NETWORK
TITLE = Set recipe parameters if starting UO_MX_CIP running SUBSTATE
//------------------------------------------------------------------------//
// Set recipe parameters:                                                 //
//------------------------------------------------------------------------//
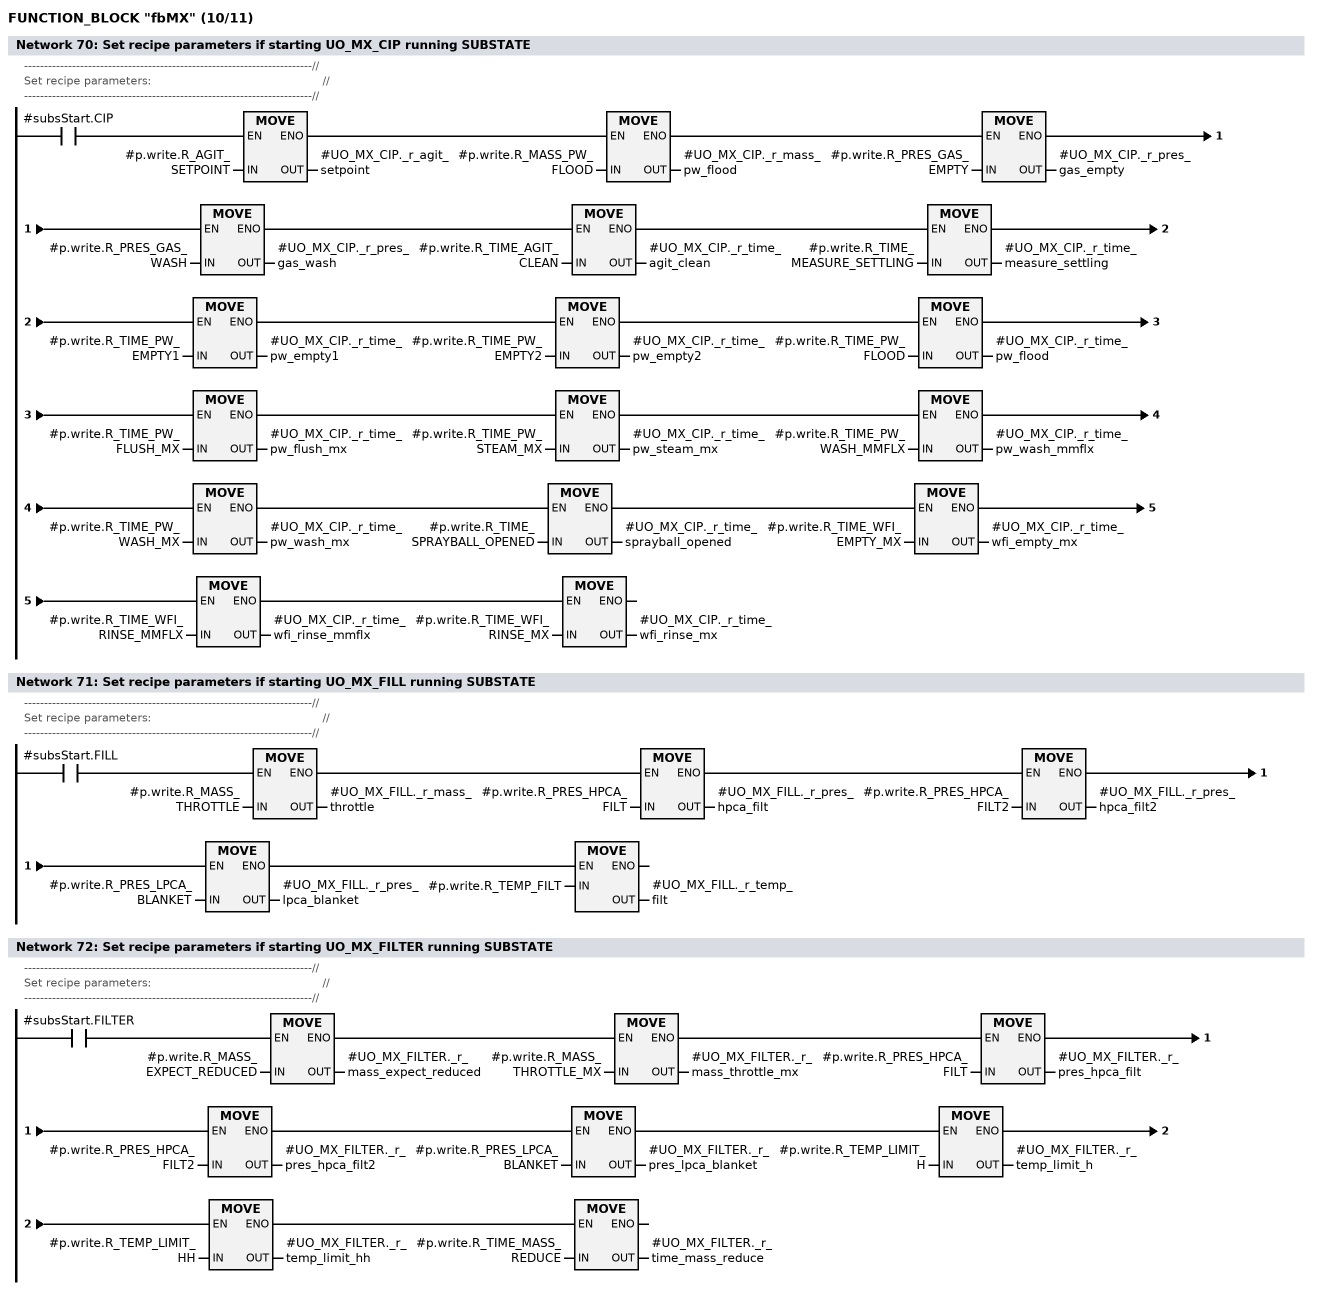
      A #subsStart.CIP;
      JCN _noStaticParms_CIP;
      L #p.write.R_AGIT_SETPOINT;
      T #UO_MX_CIP._r_agit_setpoint;
      L #p.write.R_MASS_PW_FLOOD;
      T #UO_MX_CIP._r_mass_pw_flood;
      L #p.write.R_PRES_GAS_EMPTY;
      T #UO_MX_CIP._r_pres_gas_empty;
      L #p.write.R_PRES_GAS_WASH;
      T #UO_MX_CIP._r_pres_gas_wash;
      L #p.write.R_TIME_AGIT_CLEAN;
      T #UO_MX_CIP._r_time_agit_clean;
      L #p.write.R_TIME_MEASURE_SETTLING;
      T #UO_MX_CIP._r_time_measure_settling;
      L #p.write.R_TIME_PW_EMPTY1;
      T #UO_MX_CIP._r_time_pw_empty1;
      L #p.write.R_TIME_PW_EMPTY2;
      T #UO_MX_CIP._r_time_pw_empty2;
      L #p.write.R_TIME_PW_FLOOD;
      T #UO_MX_CIP._r_time_pw_flood;
      L #p.write.R_TIME_PW_FLUSH_MX;
      T #UO_MX_CIP._r_time_pw_flush_mx;
      L #p.write.R_TIME_PW_STEAM_MX;
      T #UO_MX_CIP._r_time_pw_steam_mx;
      L #p.write.R_TIME_PW_WASH_MMFLX;
      T #UO_MX_CIP._r_time_pw_wash_mmflx;
      L #p.write.R_TIME_PW_WASH_MX;
      T #UO_MX_CIP._r_time_pw_wash_mx;
      L #p.write.R_TIME_SPRAYBALL_OPENED;
      T #UO_MX_CIP._r_time_sprayball_opened;
      L #p.write.R_TIME_WFI_EMPTY_MX;
      T #UO_MX_CIP._r_time_wfi_empty_mx;
      L #p.write.R_TIME_WFI_RINSE_MMFLX;
      T #UO_MX_CIP._r_time_wfi_rinse_mmflx;
      L #p.write.R_TIME_WFI_RINSE_MX;
      T #UO_MX_CIP._r_time_wfi_rinse_mx;

_noStaticParms_CIP:      NOP 0;
NETWORK
TITLE = Set recipe parameters if starting UO_MX_FILL running SUBSTATE
//------------------------------------------------------------------------//
// Set recipe parameters:                                                 //
//------------------------------------------------------------------------//
      A #subsStart.FILL;
      JCN _noStaticParms_FILL;
      L #p.write.R_MASS_THROTTLE;
      T #UO_MX_FILL._r_mass_throttle;
      L #p.write.R_PRES_HPCA_FILT;
      T #UO_MX_FILL._r_pres_hpca_filt;
      L #p.write.R_PRES_HPCA_FILT2;
      T #UO_MX_FILL._r_pres_hpca_filt2;
      L #p.write.R_PRES_LPCA_BLANKET;
      T #UO_MX_FILL._r_pres_lpca_blanket;
      L #p.write.R_TEMP_FILT;
      T #UO_MX_FILL._r_temp_filt;

_noStaticParms_FILL:      NOP 0;
NETWORK
TITLE = Set recipe parameters if starting UO_MX_FILTER running SUBSTATE
//------------------------------------------------------------------------//
// Set recipe parameters:                                                 //
//------------------------------------------------------------------------//
      A #subsStart.FILTER;
      JCN _noStaticParms_FILTER;
      L #p.write.R_MASS_EXPECT_REDUCED;
      T #UO_MX_FILTER._r_mass_expect_reduced;
      L #p.write.R_MASS_THROTTLE_MX;
      T #UO_MX_FILTER._r_mass_throttle_mx;
      L #p.write.R_PRES_HPCA_FILT;
      T #UO_MX_FILTER._r_pres_hpca_filt;
      L #p.write.R_PRES_HPCA_FILT2;
      T #UO_MX_FILTER._r_pres_hpca_filt2;
      L #p.write.R_PRES_LPCA_BLANKET;
      T #UO_MX_FILTER._r_pres_lpca_blanket;
      L #p.write.R_TEMP_LIMIT_H;
      T #UO_MX_FILTER._r_temp_limit_h;
      L #p.write.R_TEMP_LIMIT_HH;
      T #UO_MX_FILTER._r_temp_limit_hh;
      L #p.write.R_TIME_MASS_REDUCE;
      T #UO_MX_FILTER._r_time_mass_reduce;

_noStaticParms_FILTER:      NOP 0;
NETWORK
TITLE = Set recipe parameters if starting UO_MX_MAKE running SUBSTATE
//------------------------------------------------------------------------//
// Set recipe parameters:                                                 //
//------------------------------------------------------------------------//
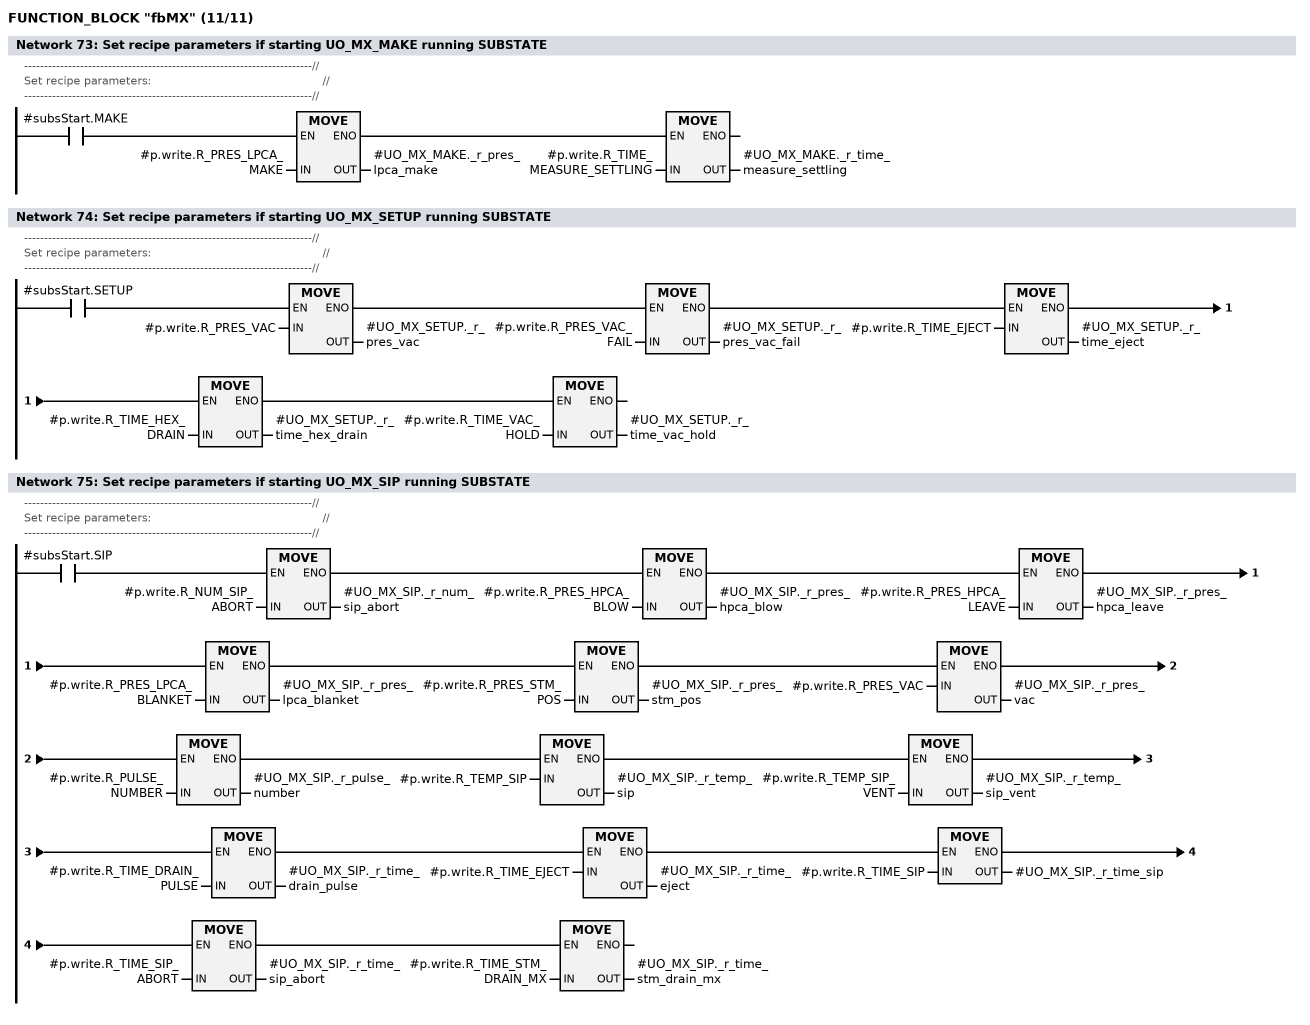
      A #subsStart.MAKE;
      JCN _noStaticParms_MAKE;
      L #p.write.R_PRES_LPCA_MAKE;
      T #UO_MX_MAKE._r_pres_lpca_make;
      L #p.write.R_TIME_MEASURE_SETTLING;
      T #UO_MX_MAKE._r_time_measure_settling;

_noStaticParms_MAKE:      NOP 0;
NETWORK
TITLE = Set recipe parameters if starting UO_MX_SETUP running SUBSTATE
//------------------------------------------------------------------------//
// Set recipe parameters:                                                 //
//------------------------------------------------------------------------//
      A #subsStart.SETUP;
      JCN _noStaticParms_SETUP;
      L #p.write.R_PRES_VAC;
      T #UO_MX_SETUP._r_pres_vac;
      L #p.write.R_PRES_VAC_FAIL;
      T #UO_MX_SETUP._r_pres_vac_fail;
      L #p.write.R_TIME_EJECT;
      T #UO_MX_SETUP._r_time_eject;
      L #p.write.R_TIME_HEX_DRAIN;
      T #UO_MX_SETUP._r_time_hex_drain;
      L #p.write.R_TIME_VAC_HOLD;
      T #UO_MX_SETUP._r_time_vac_hold;

_noStaticParms_SETUP:      NOP 0;
NETWORK
TITLE = Set recipe parameters if starting UO_MX_SIP running SUBSTATE
//------------------------------------------------------------------------//
// Set recipe parameters:                                                 //
//------------------------------------------------------------------------//
      A #subsStart.SIP;
      JCN _noStaticParms_SIP;
      L #p.write.R_NUM_SIP_ABORT;
      T #UO_MX_SIP._r_num_sip_abort;
      L #p.write.R_PRES_HPCA_BLOW;
      T #UO_MX_SIP._r_pres_hpca_blow;
      L #p.write.R_PRES_HPCA_LEAVE;
      T #UO_MX_SIP._r_pres_hpca_leave;
      L #p.write.R_PRES_LPCA_BLANKET;
      T #UO_MX_SIP._r_pres_lpca_blanket;
      L #p.write.R_PRES_STM_POS;
      T #UO_MX_SIP._r_pres_stm_pos;
      L #p.write.R_PRES_VAC;
      T #UO_MX_SIP._r_pres_vac;
      L #p.write.R_PULSE_NUMBER;
      T #UO_MX_SIP._r_pulse_number;
      L #p.write.R_TEMP_SIP;
      T #UO_MX_SIP._r_temp_sip;
      L #p.write.R_TEMP_SIP_VENT;
      T #UO_MX_SIP._r_temp_sip_vent;
      L #p.write.R_TIME_DRAIN_PULSE;
      T #UO_MX_SIP._r_time_drain_pulse;
      L #p.write.R_TIME_EJECT;
      T #UO_MX_SIP._r_time_eject;
      L #p.write.R_TIME_SIP;
      T #UO_MX_SIP._r_time_sip;
      L #p.write.R_TIME_SIP_ABORT;
      T #UO_MX_SIP._r_time_sip_abort;
      L #p.write.R_TIME_STM_DRAIN_MX;
      T #UO_MX_SIP._r_time_stm_drain_mx;

_noStaticParms_SIP:      NOP 0;

NETWORK
TITLE = Clear the operator prompt cancel flags
//------------------------------------------------------------------------//
// Clear the SFC prompt cancel flags:                                     //
//------------------------------------------------------------------------//
      R "dbEVENT".eventPrompt.event[#p.link.eventPrompt_1].cancel1;
      R "dbEVENT".eventPrompt.event[#p.link.eventPrompt_1].cancel2;
      R "dbEVENT".eventPrompt.event[#p.link.eventPrompt_1].cancel3;
      R "dbEVENT".eventPrompt.event[#p.link.eventPrompt_1].cancel4;
      R "dbEVENT".eventPrompt.event[#p.link.eventPrompt_1].cancel5;

      R "dbEVENT".eventPrompt.event[#p.link.eventPrompt_2].cancel1;
      R "dbEVENT".eventPrompt.event[#p.link.eventPrompt_2].cancel2;
      R "dbEVENT".eventPrompt.event[#p.link.eventPrompt_2].cancel3;
      R "dbEVENT".eventPrompt.event[#p.link.eventPrompt_2].cancel4;
      R "dbEVENT".eventPrompt.event[#p.link.eventPrompt_2].cancel5;

      R "dbEVENT".eventPrompt.event[#p.link.eventPrompt_3].cancel1;
      R "dbEVENT".eventPrompt.event[#p.link.eventPrompt_3].cancel2;
      R "dbEVENT".eventPrompt.event[#p.link.eventPrompt_3].cancel3;
      R "dbEVENT".eventPrompt.event[#p.link.eventPrompt_3].cancel4;
      R "dbEVENT".eventPrompt.event[#p.link.eventPrompt_3].cancel5;

      R "dbEVENT".eventPrompt.event[#p.link.eventPrompt_4].cancel1;
      R "dbEVENT".eventPrompt.event[#p.link.eventPrompt_4].cancel2;
      R "dbEVENT".eventPrompt.event[#p.link.eventPrompt_4].cancel3;
      R "dbEVENT".eventPrompt.event[#p.link.eventPrompt_4].cancel4;
      R "dbEVENT".eventPrompt.event[#p.link.eventPrompt_4].cancel5;

      R "dbEVENT".eventPrompt.event[#p.link.eventPrompt_5].cancel1;
      R "dbEVENT".eventPrompt.event[#p.link.eventPrompt_5].cancel2;
      R "dbEVENT".eventPrompt.event[#p.link.eventPrompt_5].cancel3;
      R "dbEVENT".eventPrompt.event[#p.link.eventPrompt_5].cancel4;
      R "dbEVENT".eventPrompt.event[#p.link.eventPrompt_5].cancel5;

      R "dbEVENT".eventPrompt.event[#p.link.eventPrompt_6].cancel1;
      R "dbEVENT".eventPrompt.event[#p.link.eventPrompt_6].cancel2;
      R "dbEVENT".eventPrompt.event[#p.link.eventPrompt_6].cancel3;
      R "dbEVENT".eventPrompt.event[#p.link.eventPrompt_6].cancel4;
      R "dbEVENT".eventPrompt.event[#p.link.eventPrompt_6].cancel5;

      R "dbEVENT".eventPrompt.event[#p.link.eventPrompt_7].cancel1;
      R "dbEVENT".eventPrompt.event[#p.link.eventPrompt_7].cancel2;
      R "dbEVENT".eventPrompt.event[#p.link.eventPrompt_7].cancel3;
      R "dbEVENT".eventPrompt.event[#p.link.eventPrompt_7].cancel4;
      R "dbEVENT".eventPrompt.event[#p.link.eventPrompt_7].cancel5;

      R "dbEVENT".eventPrompt.event[#p.link.eventPrompt_8].cancel1;
      R "dbEVENT".eventPrompt.event[#p.link.eventPrompt_8].cancel2;
      R "dbEVENT".eventPrompt.event[#p.link.eventPrompt_8].cancel3;
      R "dbEVENT".eventPrompt.event[#p.link.eventPrompt_8].cancel4;
      R "dbEVENT".eventPrompt.event[#p.link.eventPrompt_8].cancel5;

      R "dbEVENT".eventPrompt.event[#p.link.eventPrompt_9].cancel1;
      R "dbEVENT".eventPrompt.event[#p.link.eventPrompt_9].cancel2;
      R "dbEVENT".eventPrompt.event[#p.link.eventPrompt_9].cancel3;
      R "dbEVENT".eventPrompt.event[#p.link.eventPrompt_9].cancel4;
      R "dbEVENT".eventPrompt.event[#p.link.eventPrompt_9].cancel5;

      R "dbEVENT".eventPrompt.event[#p.link.eventPrompt_10].cancel1;
      R "dbEVENT".eventPrompt.event[#p.link.eventPrompt_10].cancel2;
      R "dbEVENT".eventPrompt.event[#p.link.eventPrompt_10].cancel3;
      R "dbEVENT".eventPrompt.event[#p.link.eventPrompt_10].cancel4;
      R "dbEVENT".eventPrompt.event[#p.link.eventPrompt_10].cancel5;

      R "dbEVENT".eventPrompt.event[#p.link.eventPrompt_11].cancel1;
      R "dbEVENT".eventPrompt.event[#p.link.eventPrompt_11].cancel2;
      R "dbEVENT".eventPrompt.event[#p.link.eventPrompt_11].cancel3;
      R "dbEVENT".eventPrompt.event[#p.link.eventPrompt_11].cancel4;
      R "dbEVENT".eventPrompt.event[#p.link.eventPrompt_11].cancel5;

      R "dbEVENT".eventPrompt.event[#p.link.eventPrompt_12].cancel1;
      R "dbEVENT".eventPrompt.event[#p.link.eventPrompt_12].cancel2;
      R "dbEVENT".eventPrompt.event[#p.link.eventPrompt_12].cancel3;
      R "dbEVENT".eventPrompt.event[#p.link.eventPrompt_12].cancel4;
      R "dbEVENT".eventPrompt.event[#p.link.eventPrompt_12].cancel5;


NETWORK
TITLE = Start the SFC sequence UO_MX_CIP in Auto for running substate CIP
//------------------------------------------------------------------------//
// START SFC   START SFC   START SFC   START SFC   START SFC   START SFC  //
//                                                                        //
// Start the running substate SFC.                                        //
//                                                                        //
// Set the running substate SFC to AUTO mode and start it:                //
//------------------------------------------------------------------------//
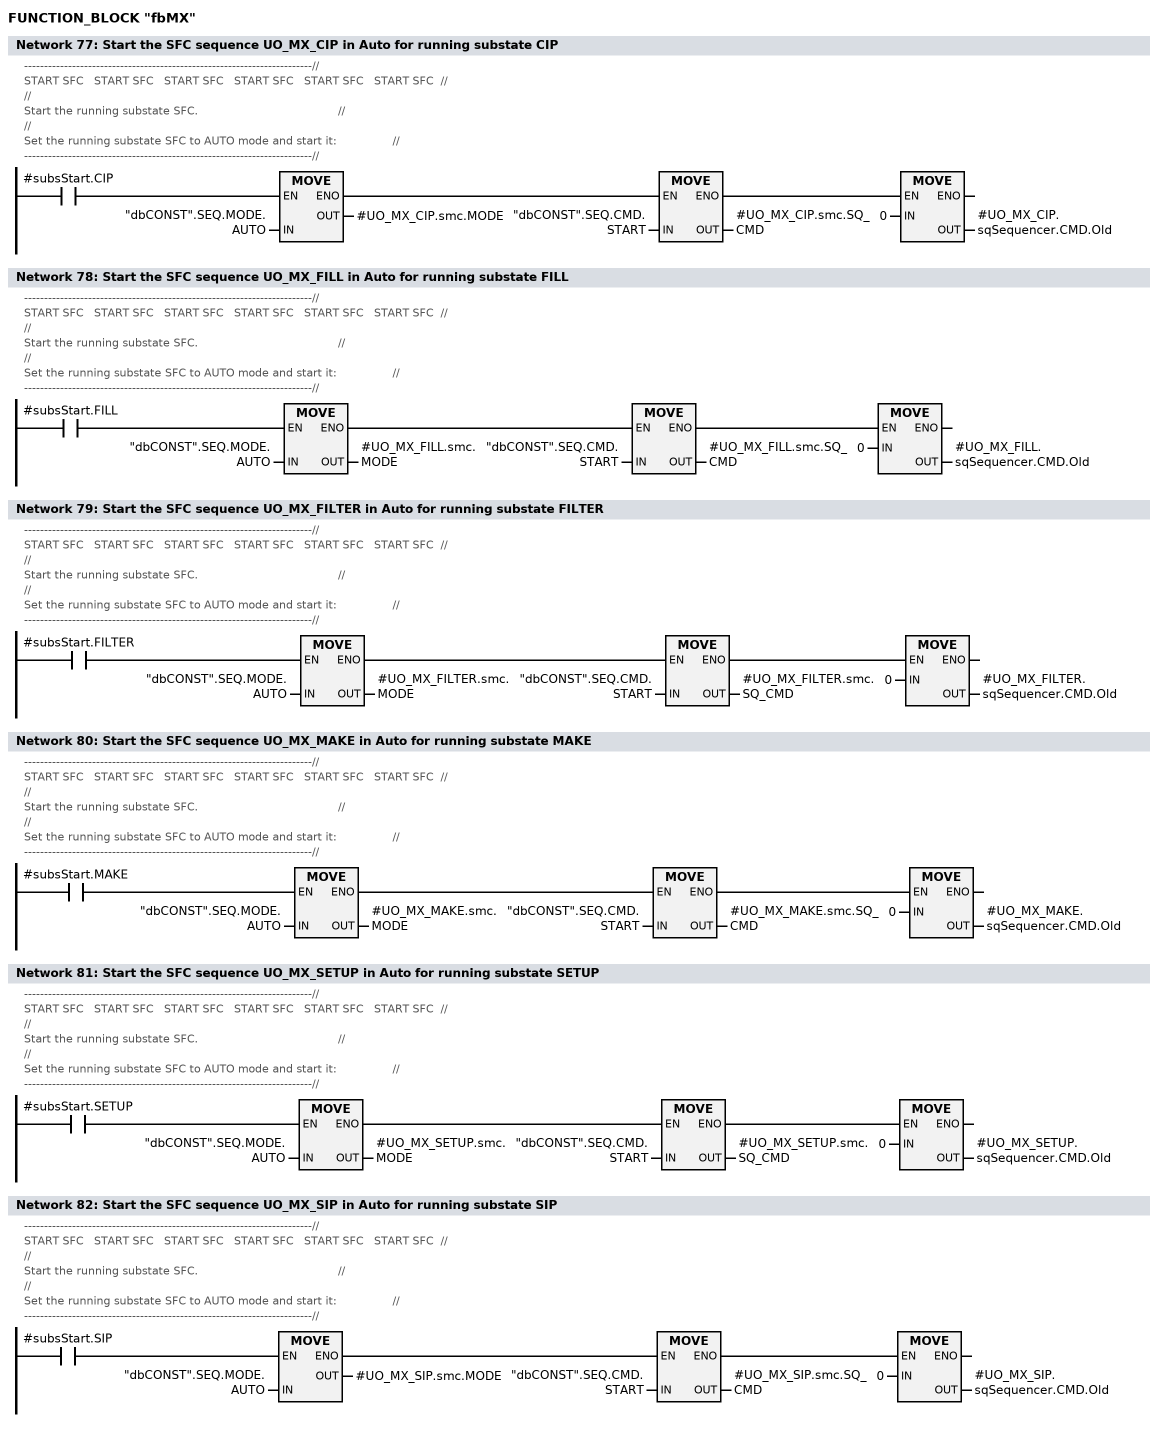
      A #subsStart.CIP;
      JCN _notSFCStarting_CIP;
      L "dbCONST".SEQ.MODE.AUTO;
      T #UO_MX_CIP.smc.MODE;
      L "dbCONST".SEQ.CMD.START;
      T #UO_MX_CIP.smc.SQ_CMD;
      L 0;
      T #UO_MX_CIP.sqSequencer.CMD.Old;

_notSFCStarting_CIP:      NOP 0;
NETWORK
TITLE = Start the SFC sequence UO_MX_FILL in Auto for running substate FILL
//------------------------------------------------------------------------//
// START SFC   START SFC   START SFC   START SFC   START SFC   START SFC  //
//                                                                        //
// Start the running substate SFC.                                        //
//                                                                        //
// Set the running substate SFC to AUTO mode and start it:                //
//------------------------------------------------------------------------//
      A #subsStart.FILL;
      JCN _notSFCStarting_FILL;
      L "dbCONST".SEQ.MODE.AUTO;
      T #UO_MX_FILL.smc.MODE;
      L "dbCONST".SEQ.CMD.START;
      T #UO_MX_FILL.smc.SQ_CMD;
      L 0;
      T #UO_MX_FILL.sqSequencer.CMD.Old;

_notSFCStarting_FILL:      NOP 0;
NETWORK
TITLE = Start the SFC sequence UO_MX_FILTER in Auto for running substate FILTER
//------------------------------------------------------------------------//
// START SFC   START SFC   START SFC   START SFC   START SFC   START SFC  //
//                                                                        //
// Start the running substate SFC.                                        //
//                                                                        //
// Set the running substate SFC to AUTO mode and start it:                //
//------------------------------------------------------------------------//
      A #subsStart.FILTER;
      JCN _notSFCStarting_FILTER;
      L "dbCONST".SEQ.MODE.AUTO;
      T #UO_MX_FILTER.smc.MODE;
      L "dbCONST".SEQ.CMD.START;
      T #UO_MX_FILTER.smc.SQ_CMD;
      L 0;
      T #UO_MX_FILTER.sqSequencer.CMD.Old;

_notSFCStarting_FILTER:      NOP 0;
NETWORK
TITLE = Start the SFC sequence UO_MX_MAKE in Auto for running substate MAKE
//------------------------------------------------------------------------//
// START SFC   START SFC   START SFC   START SFC   START SFC   START SFC  //
//                                                                        //
// Start the running substate SFC.                                        //
//                                                                        //
// Set the running substate SFC to AUTO mode and start it:                //
//------------------------------------------------------------------------//
      A #subsStart.MAKE;
      JCN _notSFCStarting_MAKE;
      L "dbCONST".SEQ.MODE.AUTO;
      T #UO_MX_MAKE.smc.MODE;
      L "dbCONST".SEQ.CMD.START;
      T #UO_MX_MAKE.smc.SQ_CMD;
      L 0;
      T #UO_MX_MAKE.sqSequencer.CMD.Old;

_notSFCStarting_MAKE:      NOP 0;
NETWORK
TITLE = Start the SFC sequence UO_MX_SETUP in Auto for running substate SETUP
//------------------------------------------------------------------------//
// START SFC   START SFC   START SFC   START SFC   START SFC   START SFC  //
//                                                                        //
// Start the running substate SFC.                                        //
//                                                                        //
// Set the running substate SFC to AUTO mode and start it:                //
//------------------------------------------------------------------------//
      A #subsStart.SETUP;
      JCN _notSFCStarting_SETUP;
      L "dbCONST".SEQ.MODE.AUTO;
      T #UO_MX_SETUP.smc.MODE;
      L "dbCONST".SEQ.CMD.START;
      T #UO_MX_SETUP.smc.SQ_CMD;
      L 0;
      T #UO_MX_SETUP.sqSequencer.CMD.Old;

_notSFCStarting_SETUP:      NOP 0;
NETWORK
TITLE = Start the SFC sequence UO_MX_SIP in Auto for running substate SIP
//------------------------------------------------------------------------//
// START SFC   START SFC   START SFC   START SFC   START SFC   START SFC  //
//                                                                        //
// Start the running substate SFC.                                        //
//                                                                        //
// Set the running substate SFC to AUTO mode and start it:                //
//------------------------------------------------------------------------//
      A #subsStart.SIP;
      JCN _notSFCStarting_SIP;
      L "dbCONST".SEQ.MODE.AUTO;
      T #UO_MX_SIP.smc.MODE;
      L "dbCONST".SEQ.CMD.START;
      T #UO_MX_SIP.smc.SQ_CMD;
      L 0;
      T #UO_MX_SIP.sqSequencer.CMD.Old;

_notSFCStarting_SIP:      NOP 0;

NETWORK
TITLE = Arm flowpath devices
//------------------------------------------------------------------------//
// Arm any flowpath child devices:                                        //
//------------------------------------------------------------------------//
      A "alwaysHigh";
      JCN _noArm_EMA_VESSEL;
      S "idbEMA1".f[#p.child.EMA_VESSEL].p.write.mc.ARMED;
_noArm_EMA_VESSEL:      NOP 0;

      A "alwaysHigh";
      JCN _noArm_EMC_GAS;
      S "idbEMC1".f[#p.child.EMC_GAS].p.write.mc.ARMED;
_noArm_EMC_GAS:      NOP 0;

      A "alwaysHigh";
      JCN _noArm_EMC_WATER;
      S "idbEMC2".f[#p.child.EMC_WATER].p.write.mc.ARMED;
_noArm_EMC_WATER:      NOP 0;

      A "alwaysHigh";
      JCN _noArm_EMG_FILTER;
      S "idbEMG1".f[#p.child.EMG_FILTER].p.write.mc.ARMED;
_noArm_EMG_FILTER:      NOP 0;

      A "alwaysHigh";
      JCN _noArm_EMM_VESSEL;
      S "idbEMM1".f[#p.child.EMM_VESSEL].p.write.mc.ARMED;
_noArm_EMM_VESSEL:      NOP 0;

      A "alwaysHigh";
      JCN _noArm_EMT_HEX;
      S "idbEMT1".f[#p.child.EMT_HEX].p.write.mc.ARMED;
_noArm_EMT_HEX:      NOP 0;

      A "alwaysHigh";
      JCN _noArm_EMV_INLET;
      S "idbEMV2".f[#p.child.EMV_INLET].p.write.mc.ARMED;
_noArm_EMV_INLET:      NOP 0;

      A "alwaysHigh";
      JCN _noArm_EMV_VESSEL;
      S "idbEMV1".f[#p.child.EMV_VESSEL].p.write.mc.ARMED;
_noArm_EMV_VESSEL:      NOP 0;

      A "alwaysHigh";
      JCN _noArm_EMX_DRAIN;
      S "idbEMX4".f[#p.child.EMX_DRAIN].p.write.mc.ARMED;
_noArm_EMX_DRAIN:      NOP 0;

      A #selected_FILL_FLZ.FL1;
      JCN _noArm_EMX_FILL1;
      S "idbEMX5".f[#p.child.EMX_FILL1].p.write.mc.ARMED;
_noArm_EMX_FILL1:      NOP 0;

      A #selected_FILL_FLZ.FL2;
      JCN _noArm_EMX_FILL2;
      S "idbEMX5".f[#p.child.EMX_FILL2].p.write.mc.ARMED;
_noArm_EMX_FILL2:      NOP 0;

      A "alwaysHigh";
      JCN _noArm_EMX_MMFL;
      S "idbEMX1".f[#p.child.EMX_MMFL].p.write.mc.ARMED;
_noArm_EMX_MMFL:      NOP 0;

      O #selected_FILL_FLZ.FL1;
      O #selected_FILL_FLZ.FL2;
      O #selected_VESSEL_SY.S1;
      O #selected_VESSEL_SY.S2;
      JCN _noArm_EMX_SMFL;
      S "idbEMX6".f[#p.child.EMX_SMFL].p.write.mc.ARMED;
_noArm_EMX_SMFL:      NOP 0;

      O #selected_FILL_FLZ.FL1;
      O #selected_FILL_FLZ.FL2;
      O #selected_VESSEL_SY.S1;
      O #selected_VESSEL_SY.S2;
      JCN _noArm_EMX_SMFLDRN;
      S "idbEMX4".f[#p.child.EMX_SMFLDRN].p.write.mc.ARMED;
_noArm_EMX_SMFLDRN:      NOP 0;

      A #selected_VESSEL_SY.S1;
      JCN _noArm_EMX_TRANSFER1;
      S "idbEMX2".f[#p.child.EMX_TRANSFER1].p.write.mc.ARMED;
_noArm_EMX_TRANSFER1:      NOP 0;

      A #selected_VESSEL_SY.S2;
      JCN _noArm_EMX_TRANSFER2;
      S "idbEMX2".f[#p.child.EMX_TRANSFER2].p.write.mc.ARMED;
_noArm_EMX_TRANSFER2:      NOP 0;


      SET;
      JC _switch_end;

  //------------------------------------------------------------------------//
  // SWITCH   SWITCH   SWITCH   SWITCH   SWITCH   SWITCH   SWITCH   SWITCH  //
  // STOPPING   STOPPING   STOPPING   STOPPING   STOPPING   STOPPING   STOP //
  // STOPPING   STOPPING   STOPPING   STOPPING   STOPPING   STOPPING   STOP //
  //------------------------------------------------------------------------//
_state_STOPPING:      NOP 0;

      SET;
      JC _switch_end;

  //------------------------------------------------------------------------//
  // SWITCH   SWITCH   SWITCH   SWITCH   SWITCH   SWITCH   SWITCH   SWITCH  //
  // RUNNING   RUNNING   RUNNING   RUNNING   RUNNING   RUNNING   RUNNING    //
  // RUNNING   RUNNING   RUNNING   RUNNING   RUNNING   RUNNING   RUNNING    //
  //------------------------------------------------------------------------//
_state_RUNNING:      NOP 0;

NETWORK
TITLE = RUNNING RUNNING RUNNING Interlock pauses the running SFC
//------------------------------------------------------------------------//
// Pause the running SFC sequence if any interlock or failure condition:  //
//------------------------------------------------------------------------//
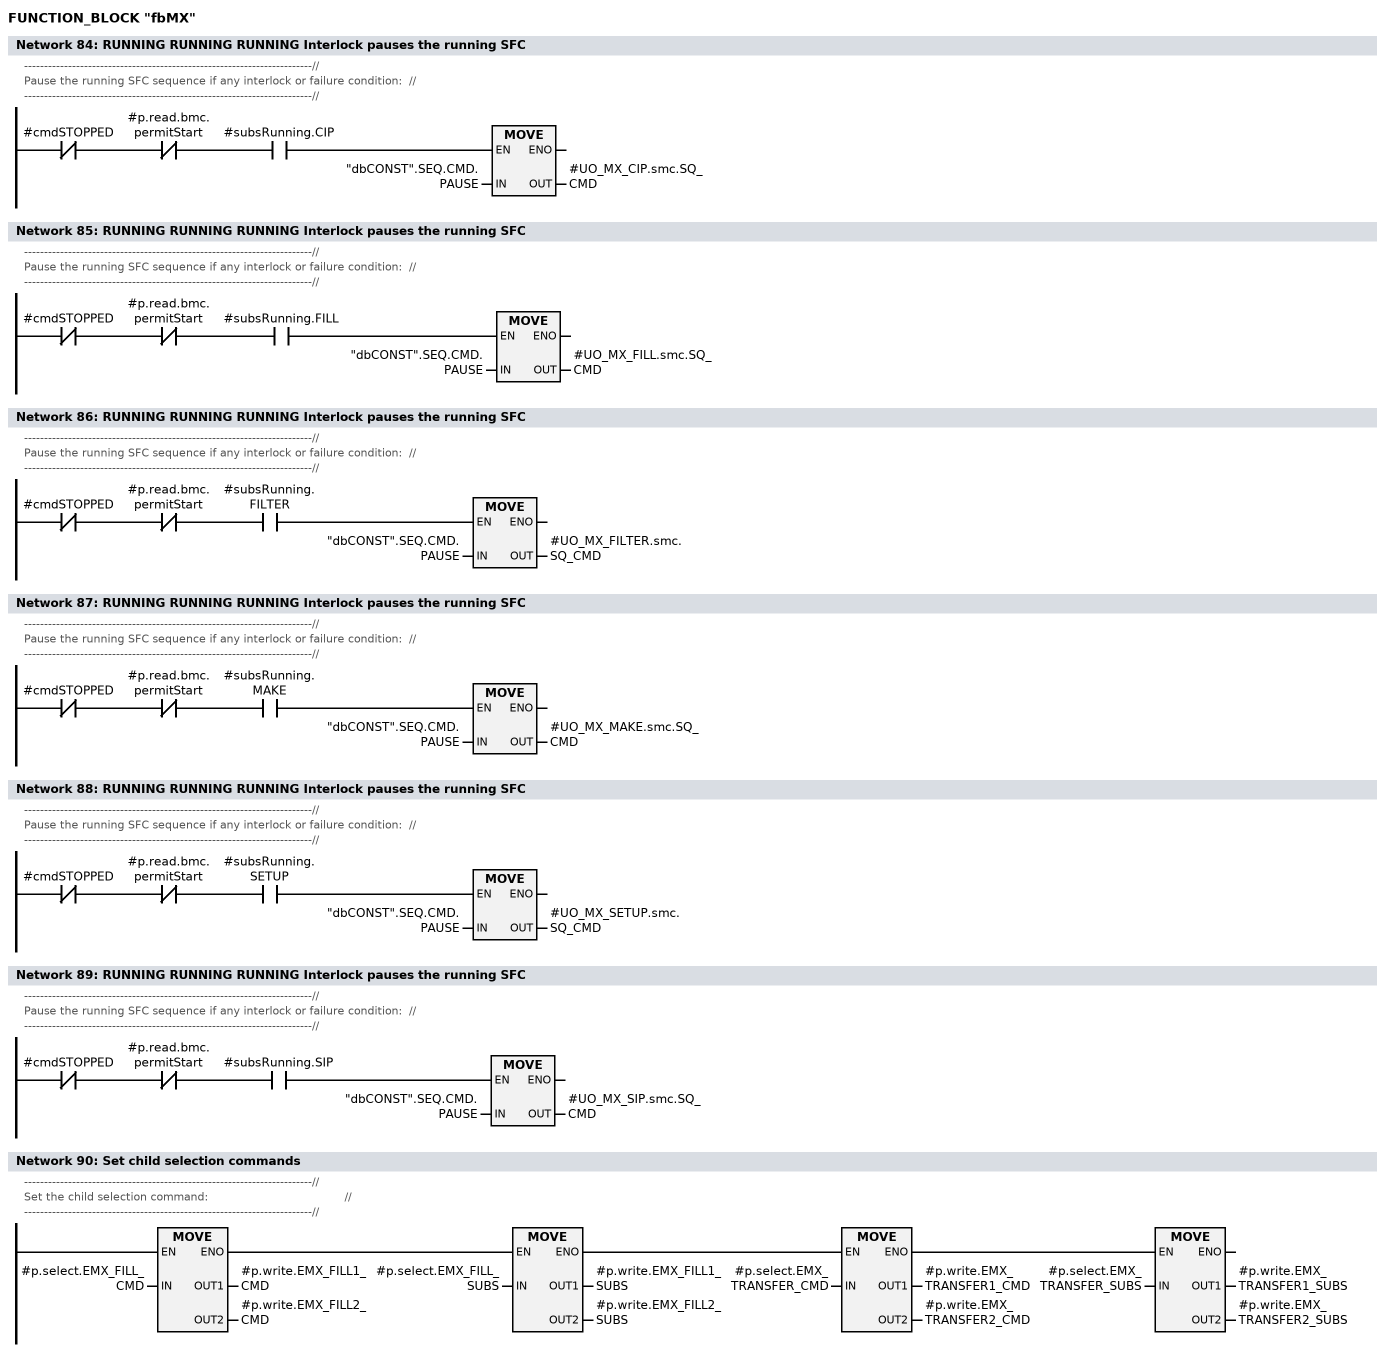
      AN #cmdSTOPPED;
      AN #p.read.bmc.permitStart;
      A #subsRunning.CIP;
      JCN _ilSFC_1;
      L "dbCONST".SEQ.CMD.PAUSE;
      T #UO_MX_CIP.smc.SQ_CMD;
_ilSFC_1:      NOP 0;

NETWORK
TITLE = RUNNING RUNNING RUNNING Interlock pauses the running SFC
//------------------------------------------------------------------------//
// Pause the running SFC sequence if any interlock or failure condition:  //
//------------------------------------------------------------------------//
      AN #cmdSTOPPED;
      AN #p.read.bmc.permitStart;
      A #subsRunning.FILL;
      JCN _ilSFC_2;
      L "dbCONST".SEQ.CMD.PAUSE;
      T #UO_MX_FILL.smc.SQ_CMD;
_ilSFC_2:      NOP 0;

NETWORK
TITLE = RUNNING RUNNING RUNNING Interlock pauses the running SFC
//------------------------------------------------------------------------//
// Pause the running SFC sequence if any interlock or failure condition:  //
//------------------------------------------------------------------------//
      AN #cmdSTOPPED;
      AN #p.read.bmc.permitStart;
      A #subsRunning.FILTER;
      JCN _ilSFC_3;
      L "dbCONST".SEQ.CMD.PAUSE;
      T #UO_MX_FILTER.smc.SQ_CMD;
_ilSFC_3:      NOP 0;

NETWORK
TITLE = RUNNING RUNNING RUNNING Interlock pauses the running SFC
//------------------------------------------------------------------------//
// Pause the running SFC sequence if any interlock or failure condition:  //
//------------------------------------------------------------------------//
      AN #cmdSTOPPED;
      AN #p.read.bmc.permitStart;
      A #subsRunning.MAKE;
      JCN _ilSFC_4;
      L "dbCONST".SEQ.CMD.PAUSE;
      T #UO_MX_MAKE.smc.SQ_CMD;
_ilSFC_4:      NOP 0;

NETWORK
TITLE = RUNNING RUNNING RUNNING Interlock pauses the running SFC
//------------------------------------------------------------------------//
// Pause the running SFC sequence if any interlock or failure condition:  //
//------------------------------------------------------------------------//
      AN #cmdSTOPPED;
      AN #p.read.bmc.permitStart;
      A #subsRunning.SETUP;
      JCN _ilSFC_5;
      L "dbCONST".SEQ.CMD.PAUSE;
      T #UO_MX_SETUP.smc.SQ_CMD;
_ilSFC_5:      NOP 0;

NETWORK
TITLE = RUNNING RUNNING RUNNING Interlock pauses the running SFC
//------------------------------------------------------------------------//
// Pause the running SFC sequence if any interlock or failure condition:  //
//------------------------------------------------------------------------//
      AN #cmdSTOPPED;
      AN #p.read.bmc.permitStart;
      A #subsRunning.SIP;
      JCN _ilSFC_6;
      L "dbCONST".SEQ.CMD.PAUSE;
      T #UO_MX_SIP.smc.SQ_CMD;
_ilSFC_6:      NOP 0;


NETWORK
TITLE = Set child selection commands
//------------------------------------------------------------------------//
// Set the child selection command:                                       //
//------------------------------------------------------------------------//
      L #p.select.EMX_FILL_CMD;
      T #p.write.EMX_FILL1_CMD;
      T #p.write.EMX_FILL2_CMD;
      L #p.select.EMX_FILL_SUBS;
      T #p.write.EMX_FILL1_SUBS;
      T #p.write.EMX_FILL2_SUBS;
      L #p.select.EMX_TRANSFER_CMD;
      T #p.write.EMX_TRANSFER1_CMD;
      T #p.write.EMX_TRANSFER2_CMD;
      L #p.select.EMX_TRANSFER_SUBS;
      T #p.write.EMX_TRANSFER1_SUBS;
      T #p.write.EMX_TRANSFER2_SUBS;

NETWORK
TITLE = Set the child command attributes
//------------------------------------------------------------------------//
// Upload the child state:                                                //
//------------------------------------------------------------------------//


NETWORK
TITLE = Raise operator prompt if required
//------------------------------------------------------------------------//
// OPERATOR PROMPT   OPERATOR PROMPT   OPERATOR PROMPT   OPERATOR PROMPT  //
//                                                                        //
// Transfer the SFC eventPrompt bit to the global event datablock:        //
//------------------------------------------------------------------------//
      O #subsRunning.CIP;
      O #subsRunning.FILL;
      O #subsRunning.FILTER;
      O #subsRunning.MAKE;
      O #subsRunning.SETUP;
      O #subsRunning.SIP;
      JCN _noRunPrompt;

      A #UO_MX_FILL._prompt_abort;
      JCN _not_eventPrompt_31;
      L #p.write.mc.SERIALNUM;
      T "dbEVENT".eventPrompt.event[#p.link.eventPrompt_1].numSerial;
      R #UO_MX_FILL._prompt_abort;
      R "dbEVENT".eventPrompt.event[#p.link.eventPrompt_1].confirmYes;
      R "dbEVENT".eventPrompt.event[#p.link.eventPrompt_1].confirmNo;
      S "dbEVENT".eventPrompt.event[#p.link.eventPrompt_1].trigger1;
      S "dbEVENT".eventPrompt.event[#p.link.eventPrompt_1].trigger2;
      S "dbEVENT".eventPrompt.event[#p.link.eventPrompt_1].trigger3;
      S "dbEVENT".eventPrompt.event[#p.link.eventPrompt_1].trigger4;
      S "dbEVENT".eventPrompt.event[#p.link.eventPrompt_1].trigger5;
_not_eventPrompt_31:      NOP 0;

      A #UO_MX_FILTER._prompt_abort;
      JCN _not_eventPrompt_32;
      L #p.write.mc.SERIALNUM;
      T "dbEVENT".eventPrompt.event[#p.link.eventPrompt_2].numSerial;
      R #UO_MX_FILTER._prompt_abort;
      R "dbEVENT".eventPrompt.event[#p.link.eventPrompt_2].confirmYes;
      R "dbEVENT".eventPrompt.event[#p.link.eventPrompt_2].confirmNo;
      S "dbEVENT".eventPrompt.event[#p.link.eventPrompt_2].trigger1;
      S "dbEVENT".eventPrompt.event[#p.link.eventPrompt_2].trigger2;
      S "dbEVENT".eventPrompt.event[#p.link.eventPrompt_2].trigger3;
      S "dbEVENT".eventPrompt.event[#p.link.eventPrompt_2].trigger4;
      S "dbEVENT".eventPrompt.event[#p.link.eventPrompt_2].trigger5;
_not_eventPrompt_32:      NOP 0;

      A #UO_MX_SETUP._prompt_connect_ok;
      JCN _not_eventPrompt_33;
      L #p.write.mc.SERIALNUM;
      T "dbEVENT".eventPrompt.event[#p.link.eventPrompt_3].numSerial;
      R #UO_MX_SETUP._prompt_connect_ok;
      R "dbEVENT".eventPrompt.event[#p.link.eventPrompt_3].confirmYes;
      R "dbEVENT".eventPrompt.event[#p.link.eventPrompt_3].confirmNo;
      S "dbEVENT".eventPrompt.event[#p.link.eventPrompt_3].trigger1;
      S "dbEVENT".eventPrompt.event[#p.link.eventPrompt_3].trigger2;
      S "dbEVENT".eventPrompt.event[#p.link.eventPrompt_3].trigger3;
      S "dbEVENT".eventPrompt.event[#p.link.eventPrompt_3].trigger4;
      S "dbEVENT".eventPrompt.event[#p.link.eventPrompt_3].trigger5;
_not_eventPrompt_33:      NOP 0;

      A #UO_MX_FILTER._prompt_filt_completed;
      JCN _not_eventPrompt_34;
      L #p.write.mc.SERIALNUM;
      T "dbEVENT".eventPrompt.event[#p.link.eventPrompt_4].numSerial;
      R #UO_MX_FILTER._prompt_filt_completed;
      R "dbEVENT".eventPrompt.event[#p.link.eventPrompt_4].confirmYes;
      R "dbEVENT".eventPrompt.event[#p.link.eventPrompt_4].confirmNo;
      S "dbEVENT".eventPrompt.event[#p.link.eventPrompt_4].trigger1;
      S "dbEVENT".eventPrompt.event[#p.link.eventPrompt_4].trigger2;
      S "dbEVENT".eventPrompt.event[#p.link.eventPrompt_4].trigger3;
      S "dbEVENT".eventPrompt.event[#p.link.eventPrompt_4].trigger4;
      S "dbEVENT".eventPrompt.event[#p.link.eventPrompt_4].trigger5;
_not_eventPrompt_34:      NOP 0;

      A #UO_MX_FILL._prompt_filtration;
      JCN _not_eventPrompt_35;
      L #p.write.mc.SERIALNUM;
      T "dbEVENT".eventPrompt.event[#p.link.eventPrompt_5].numSerial;
      R #UO_MX_FILL._prompt_filtration;
      R "dbEVENT".eventPrompt.event[#p.link.eventPrompt_5].confirmYes;
      R "dbEVENT".eventPrompt.event[#p.link.eventPrompt_5].confirmNo;
      S "dbEVENT".eventPrompt.event[#p.link.eventPrompt_5].trigger1;
      S "dbEVENT".eventPrompt.event[#p.link.eventPrompt_5].trigger2;
      S "dbEVENT".eventPrompt.event[#p.link.eventPrompt_5].trigger3;
      S "dbEVENT".eventPrompt.event[#p.link.eventPrompt_5].trigger4;
      S "dbEVENT".eventPrompt.event[#p.link.eventPrompt_5].trigger5;
_not_eventPrompt_35:      NOP 0;

      A #UO_MX_FILTER._prompt_filtration;
      JCN _not_eventPrompt_36;
      L #p.write.mc.SERIALNUM;
      T "dbEVENT".eventPrompt.event[#p.link.eventPrompt_6].numSerial;
      R #UO_MX_FILTER._prompt_filtration;
      R "dbEVENT".eventPrompt.event[#p.link.eventPrompt_6].confirmYes;
      R "dbEVENT".eventPrompt.event[#p.link.eventPrompt_6].confirmNo;
      S "dbEVENT".eventPrompt.event[#p.link.eventPrompt_6].trigger1;
      S "dbEVENT".eventPrompt.event[#p.link.eventPrompt_6].trigger2;
      S "dbEVENT".eventPrompt.event[#p.link.eventPrompt_6].trigger3;
      S "dbEVENT".eventPrompt.event[#p.link.eventPrompt_6].trigger4;
      S "dbEVENT".eventPrompt.event[#p.link.eventPrompt_6].trigger5;
_not_eventPrompt_36:      NOP 0;

      A #UO_MX_MAKE._prompt_manway_complete;
      JCN _not_eventPrompt_37;
      L #p.write.mc.SERIALNUM;
      T "dbEVENT".eventPrompt.event[#p.link.eventPrompt_7].numSerial;
      R #UO_MX_MAKE._prompt_manway_complete;
      R "dbEVENT".eventPrompt.event[#p.link.eventPrompt_7].confirmYes;
      R "dbEVENT".eventPrompt.event[#p.link.eventPrompt_7].confirmNo;
      S "dbEVENT".eventPrompt.event[#p.link.eventPrompt_7].trigger1;
      S "dbEVENT".eventPrompt.event[#p.link.eventPrompt_7].trigger2;
      S "dbEVENT".eventPrompt.event[#p.link.eventPrompt_7].trigger3;
      S "dbEVENT".eventPrompt.event[#p.link.eventPrompt_7].trigger4;
      S "dbEVENT".eventPrompt.event[#p.link.eventPrompt_7].trigger5;
_not_eventPrompt_37:      NOP 0;

      A #UO_MX_SETUP._prompt_not_held;
      JCN _not_eventPrompt_38;
      L #p.write.mc.SERIALNUM;
      T "dbEVENT".eventPrompt.event[#p.link.eventPrompt_8].numSerial;
      R #UO_MX_SETUP._prompt_not_held;
      R "dbEVENT".eventPrompt.event[#p.link.eventPrompt_8].confirmYes;
      R "dbEVENT".eventPrompt.event[#p.link.eventPrompt_8].confirmNo;
      S "dbEVENT".eventPrompt.event[#p.link.eventPrompt_8].trigger1;
      S "dbEVENT".eventPrompt.event[#p.link.eventPrompt_8].trigger2;
      S "dbEVENT".eventPrompt.event[#p.link.eventPrompt_8].trigger3;
      S "dbEVENT".eventPrompt.event[#p.link.eventPrompt_8].trigger4;
      S "dbEVENT".eventPrompt.event[#p.link.eventPrompt_8].trigger5;
_not_eventPrompt_38:      NOP 0;

      A #UO_MX_SETUP._prompt_not_reach;
      JCN _not_eventPrompt_39;
      L #p.write.mc.SERIALNUM;
      T "dbEVENT".eventPrompt.event[#p.link.eventPrompt_9].numSerial;
      R #UO_MX_SETUP._prompt_not_reach;
      R "dbEVENT".eventPrompt.event[#p.link.eventPrompt_9].confirmYes;
      R "dbEVENT".eventPrompt.event[#p.link.eventPrompt_9].confirmNo;
      S "dbEVENT".eventPrompt.event[#p.link.eventPrompt_9].trigger1;
      S "dbEVENT".eventPrompt.event[#p.link.eventPrompt_9].trigger2;
      S "dbEVENT".eventPrompt.event[#p.link.eventPrompt_9].trigger3;
      S "dbEVENT".eventPrompt.event[#p.link.eventPrompt_9].trigger4;
      S "dbEVENT".eventPrompt.event[#p.link.eventPrompt_9].trigger5;
_not_eventPrompt_39:      NOP 0;

      A #UO_MX_MAKE._prompt_pmo;
      JCN _not_eventPrompt_40;
      L #p.write.mc.SERIALNUM;
      T "dbEVENT".eventPrompt.event[#p.link.eventPrompt_10].numSerial;
      R #UO_MX_MAKE._prompt_pmo;
      R "dbEVENT".eventPrompt.event[#p.link.eventPrompt_10].confirmYes;
      R "dbEVENT".eventPrompt.event[#p.link.eventPrompt_10].confirmNo;
      S "dbEVENT".eventPrompt.event[#p.link.eventPrompt_10].trigger1;
      S "dbEVENT".eventPrompt.event[#p.link.eventPrompt_10].trigger2;
      S "dbEVENT".eventPrompt.event[#p.link.eventPrompt_10].trigger3;
      S "dbEVENT".eventPrompt.event[#p.link.eventPrompt_10].trigger4;
      S "dbEVENT".eventPrompt.event[#p.link.eventPrompt_10].trigger5;
_not_eventPrompt_40:      NOP 0;

      A #UO_MX_MAKE._prompt_tare;
      JCN _not_eventPrompt_41;
      L #p.write.mc.SERIALNUM;
      T "dbEVENT".eventPrompt.event[#p.link.eventPrompt_11].numSerial;
      R #UO_MX_MAKE._prompt_tare;
      R "dbEVENT".eventPrompt.event[#p.link.eventPrompt_11].confirmYes;
      R "dbEVENT".eventPrompt.event[#p.link.eventPrompt_11].confirmNo;
      S "dbEVENT".eventPrompt.event[#p.link.eventPrompt_11].trigger1;
      S "dbEVENT".eventPrompt.event[#p.link.eventPrompt_11].trigger2;
      S "dbEVENT".eventPrompt.event[#p.link.eventPrompt_11].trigger3;
      S "dbEVENT".eventPrompt.event[#p.link.eventPrompt_11].trigger4;
      S "dbEVENT".eventPrompt.event[#p.link.eventPrompt_11].trigger5;
_not_eventPrompt_41:      NOP 0;

      A #UO_MX_SIP._prompt_try_again;
      JCN _not_eventPrompt_42;
      L #p.write.mc.SERIALNUM;
      T "dbEVENT".eventPrompt.event[#p.link.eventPrompt_12].numSerial;
      R #UO_MX_SIP._prompt_try_again;
      R "dbEVENT".eventPrompt.event[#p.link.eventPrompt_12].confirmYes;
      R "dbEVENT".eventPrompt.event[#p.link.eventPrompt_12].confirmNo;
      S "dbEVENT".eventPrompt.event[#p.link.eventPrompt_12].trigger1;
      S "dbEVENT".eventPrompt.event[#p.link.eventPrompt_12].trigger2;
      S "dbEVENT".eventPrompt.event[#p.link.eventPrompt_12].trigger3;
      S "dbEVENT".eventPrompt.event[#p.link.eventPrompt_12].trigger4;
      S "dbEVENT".eventPrompt.event[#p.link.eventPrompt_12].trigger5;
_not_eventPrompt_42:      NOP 0;

_noRunPrompt:      NOP 0;

NETWORK
TITLE = Check if operator confirm bit response
//------------------------------------------------------------------------//
// OPERATOR CONFIRM   OPERATOR CONFIRM   OPERATOR CONFIRM   OPERATOR CONF //
//                                                                        //
// Check if a confirm response has been received:                         //
//------------------------------------------------------------------------//
      O "dbEVENT".eventPrompt.event[#p.link.eventPrompt_1].confirmYes;
      O "dbEVENT".eventPrompt.event[#p.link.eventPrompt_1].confirmNo;
      JCN _not_eventPrompt_31_response;
      R "dbEVENT".eventPrompt.event[#p.link.eventPrompt_1].trigger1;
      R "dbEVENT".eventPrompt.event[#p.link.eventPrompt_1].trigger2;
      R "dbEVENT".eventPrompt.event[#p.link.eventPrompt_1].trigger3;
      R "dbEVENT".eventPrompt.event[#p.link.eventPrompt_1].trigger4;
      R "dbEVENT".eventPrompt.event[#p.link.eventPrompt_1].trigger5;
      S "dbEVENT".eventPrompt.event[#p.link.eventPrompt_1].cancel1;
      S "dbEVENT".eventPrompt.event[#p.link.eventPrompt_1].cancel2;
      S "dbEVENT".eventPrompt.event[#p.link.eventPrompt_1].cancel3;
      S "dbEVENT".eventPrompt.event[#p.link.eventPrompt_1].cancel4;
      S "dbEVENT".eventPrompt.event[#p.link.eventPrompt_1].cancel5;
_not_eventPrompt_31_response:      NOP 0;

      O "dbEVENT".eventPrompt.event[#p.link.eventPrompt_2].confirmYes;
      O "dbEVENT".eventPrompt.event[#p.link.eventPrompt_2].confirmNo;
      JCN _not_eventPrompt_32_response;
      R "dbEVENT".eventPrompt.event[#p.link.eventPrompt_2].trigger1;
      R "dbEVENT".eventPrompt.event[#p.link.eventPrompt_2].trigger2;
      R "dbEVENT".eventPrompt.event[#p.link.eventPrompt_2].trigger3;
      R "dbEVENT".eventPrompt.event[#p.link.eventPrompt_2].trigger4;
      R "dbEVENT".eventPrompt.event[#p.link.eventPrompt_2].trigger5;
      S "dbEVENT".eventPrompt.event[#p.link.eventPrompt_2].cancel1;
      S "dbEVENT".eventPrompt.event[#p.link.eventPrompt_2].cancel2;
      S "dbEVENT".eventPrompt.event[#p.link.eventPrompt_2].cancel3;
      S "dbEVENT".eventPrompt.event[#p.link.eventPrompt_2].cancel4;
      S "dbEVENT".eventPrompt.event[#p.link.eventPrompt_2].cancel5;
_not_eventPrompt_32_response:      NOP 0;

      O "dbEVENT".eventPrompt.event[#p.link.eventPrompt_3].confirmYes;
      O "dbEVENT".eventPrompt.event[#p.link.eventPrompt_3].confirmNo;
      JCN _not_eventPrompt_33_response;
      R "dbEVENT".eventPrompt.event[#p.link.eventPrompt_3].trigger1;
      R "dbEVENT".eventPrompt.event[#p.link.eventPrompt_3].trigger2;
      R "dbEVENT".eventPrompt.event[#p.link.eventPrompt_3].trigger3;
      R "dbEVENT".eventPrompt.event[#p.link.eventPrompt_3].trigger4;
      R "dbEVENT".eventPrompt.event[#p.link.eventPrompt_3].trigger5;
      S "dbEVENT".eventPrompt.event[#p.link.eventPrompt_3].cancel1;
      S "dbEVENT".eventPrompt.event[#p.link.eventPrompt_3].cancel2;
      S "dbEVENT".eventPrompt.event[#p.link.eventPrompt_3].cancel3;
      S "dbEVENT".eventPrompt.event[#p.link.eventPrompt_3].cancel4;
      S "dbEVENT".eventPrompt.event[#p.link.eventPrompt_3].cancel5;
_not_eventPrompt_33_response:      NOP 0;

      O "dbEVENT".eventPrompt.event[#p.link.eventPrompt_4].confirmYes;
      O "dbEVENT".eventPrompt.event[#p.link.eventPrompt_4].confirmNo;
      JCN _not_eventPrompt_34_response;
      R "dbEVENT".eventPrompt.event[#p.link.eventPrompt_4].trigger1;
      R "dbEVENT".eventPrompt.event[#p.link.eventPrompt_4].trigger2;
      R "dbEVENT".eventPrompt.event[#p.link.eventPrompt_4].trigger3;
      R "dbEVENT".eventPrompt.event[#p.link.eventPrompt_4].trigger4;
      R "dbEVENT".eventPrompt.event[#p.link.eventPrompt_4].trigger5;
      S "dbEVENT".eventPrompt.event[#p.link.eventPrompt_4].cancel1;
      S "dbEVENT".eventPrompt.event[#p.link.eventPrompt_4].cancel2;
      S "dbEVENT".eventPrompt.event[#p.link.eventPrompt_4].cancel3;
      S "dbEVENT".eventPrompt.event[#p.link.eventPrompt_4].cancel4;
      S "dbEVENT".eventPrompt.event[#p.link.eventPrompt_4].cancel5;
_not_eventPrompt_34_response:      NOP 0;

      O "dbEVENT".eventPrompt.event[#p.link.eventPrompt_5].confirmYes;
      O "dbEVENT".eventPrompt.event[#p.link.eventPrompt_5].confirmNo;
      JCN _not_eventPrompt_35_response;
      R "dbEVENT".eventPrompt.event[#p.link.eventPrompt_5].trigger1;
      R "dbEVENT".eventPrompt.event[#p.link.eventPrompt_5].trigger2;
      R "dbEVENT".eventPrompt.event[#p.link.eventPrompt_5].trigger3;
      R "dbEVENT".eventPrompt.event[#p.link.eventPrompt_5].trigger4;
      R "dbEVENT".eventPrompt.event[#p.link.eventPrompt_5].trigger5;
      S "dbEVENT".eventPrompt.event[#p.link.eventPrompt_5].cancel1;
      S "dbEVENT".eventPrompt.event[#p.link.eventPrompt_5].cancel2;
      S "dbEVENT".eventPrompt.event[#p.link.eventPrompt_5].cancel3;
      S "dbEVENT".eventPrompt.event[#p.link.eventPrompt_5].cancel4;
      S "dbEVENT".eventPrompt.event[#p.link.eventPrompt_5].cancel5;
_not_eventPrompt_35_response:      NOP 0;

      O "dbEVENT".eventPrompt.event[#p.link.eventPrompt_6].confirmYes;
      O "dbEVENT".eventPrompt.event[#p.link.eventPrompt_6].confirmNo;
      JCN _not_eventPrompt_36_response;
      R "dbEVENT".eventPrompt.event[#p.link.eventPrompt_6].trigger1;
      R "dbEVENT".eventPrompt.event[#p.link.eventPrompt_6].trigger2;
      R "dbEVENT".eventPrompt.event[#p.link.eventPrompt_6].trigger3;
      R "dbEVENT".eventPrompt.event[#p.link.eventPrompt_6].trigger4;
      R "dbEVENT".eventPrompt.event[#p.link.eventPrompt_6].trigger5;
      S "dbEVENT".eventPrompt.event[#p.link.eventPrompt_6].cancel1;
      S "dbEVENT".eventPrompt.event[#p.link.eventPrompt_6].cancel2;
      S "dbEVENT".eventPrompt.event[#p.link.eventPrompt_6].cancel3;
      S "dbEVENT".eventPrompt.event[#p.link.eventPrompt_6].cancel4;
      S "dbEVENT".eventPrompt.event[#p.link.eventPrompt_6].cancel5;
_not_eventPrompt_36_response:      NOP 0;

      O "dbEVENT".eventPrompt.event[#p.link.eventPrompt_7].confirmYes;
      O "dbEVENT".eventPrompt.event[#p.link.eventPrompt_7].confirmNo;
      JCN _not_eventPrompt_37_response;
      R "dbEVENT".eventPrompt.event[#p.link.eventPrompt_7].trigger1;
      R "dbEVENT".eventPrompt.event[#p.link.eventPrompt_7].trigger2;
      R "dbEVENT".eventPrompt.event[#p.link.eventPrompt_7].trigger3;
      R "dbEVENT".eventPrompt.event[#p.link.eventPrompt_7].trigger4;
      R "dbEVENT".eventPrompt.event[#p.link.eventPrompt_7].trigger5;
      S "dbEVENT".eventPrompt.event[#p.link.eventPrompt_7].cancel1;
      S "dbEVENT".eventPrompt.event[#p.link.eventPrompt_7].cancel2;
      S "dbEVENT".eventPrompt.event[#p.link.eventPrompt_7].cancel3;
      S "dbEVENT".eventPrompt.event[#p.link.eventPrompt_7].cancel4;
      S "dbEVENT".eventPrompt.event[#p.link.eventPrompt_7].cancel5;
_not_eventPrompt_37_response:      NOP 0;

      O "dbEVENT".eventPrompt.event[#p.link.eventPrompt_8].confirmYes;
      O "dbEVENT".eventPrompt.event[#p.link.eventPrompt_8].confirmNo;
      JCN _not_eventPrompt_38_response;
      R "dbEVENT".eventPrompt.event[#p.link.eventPrompt_8].trigger1;
      R "dbEVENT".eventPrompt.event[#p.link.eventPrompt_8].trigger2;
      R "dbEVENT".eventPrompt.event[#p.link.eventPrompt_8].trigger3;
      R "dbEVENT".eventPrompt.event[#p.link.eventPrompt_8].trigger4;
      R "dbEVENT".eventPrompt.event[#p.link.eventPrompt_8].trigger5;
      S "dbEVENT".eventPrompt.event[#p.link.eventPrompt_8].cancel1;
      S "dbEVENT".eventPrompt.event[#p.link.eventPrompt_8].cancel2;
      S "dbEVENT".eventPrompt.event[#p.link.eventPrompt_8].cancel3;
      S "dbEVENT".eventPrompt.event[#p.link.eventPrompt_8].cancel4;
      S "dbEVENT".eventPrompt.event[#p.link.eventPrompt_8].cancel5;
_not_eventPrompt_38_response:      NOP 0;

      O "dbEVENT".eventPrompt.event[#p.link.eventPrompt_9].confirmYes;
      O "dbEVENT".eventPrompt.event[#p.link.eventPrompt_9].confirmNo;
      JCN _not_eventPrompt_39_response;
      R "dbEVENT".eventPrompt.event[#p.link.eventPrompt_9].trigger1;
      R "dbEVENT".eventPrompt.event[#p.link.eventPrompt_9].trigger2;
      R "dbEVENT".eventPrompt.event[#p.link.eventPrompt_9].trigger3;
      R "dbEVENT".eventPrompt.event[#p.link.eventPrompt_9].trigger4;
      R "dbEVENT".eventPrompt.event[#p.link.eventPrompt_9].trigger5;
      S "dbEVENT".eventPrompt.event[#p.link.eventPrompt_9].cancel1;
      S "dbEVENT".eventPrompt.event[#p.link.eventPrompt_9].cancel2;
      S "dbEVENT".eventPrompt.event[#p.link.eventPrompt_9].cancel3;
      S "dbEVENT".eventPrompt.event[#p.link.eventPrompt_9].cancel4;
      S "dbEVENT".eventPrompt.event[#p.link.eventPrompt_9].cancel5;
_not_eventPrompt_39_response:      NOP 0;

      O "dbEVENT".eventPrompt.event[#p.link.eventPrompt_10].confirmYes;
      O "dbEVENT".eventPrompt.event[#p.link.eventPrompt_10].confirmNo;
      JCN _not_eventPrompt_40_response;
      R "dbEVENT".eventPrompt.event[#p.link.eventPrompt_10].trigger1;
      R "dbEVENT".eventPrompt.event[#p.link.eventPrompt_10].trigger2;
      R "dbEVENT".eventPrompt.event[#p.link.eventPrompt_10].trigger3;
      R "dbEVENT".eventPrompt.event[#p.link.eventPrompt_10].trigger4;
      R "dbEVENT".eventPrompt.event[#p.link.eventPrompt_10].trigger5;
      S "dbEVENT".eventPrompt.event[#p.link.eventPrompt_10].cancel1;
      S "dbEVENT".eventPrompt.event[#p.link.eventPrompt_10].cancel2;
      S "dbEVENT".eventPrompt.event[#p.link.eventPrompt_10].cancel3;
      S "dbEVENT".eventPrompt.event[#p.link.eventPrompt_10].cancel4;
      S "dbEVENT".eventPrompt.event[#p.link.eventPrompt_10].cancel5;
_not_eventPrompt_40_response:      NOP 0;

      O "dbEVENT".eventPrompt.event[#p.link.eventPrompt_11].confirmYes;
      O "dbEVENT".eventPrompt.event[#p.link.eventPrompt_11].confirmNo;
      JCN _not_eventPrompt_41_response;
      R "dbEVENT".eventPrompt.event[#p.link.eventPrompt_11].trigger1;
      R "dbEVENT".eventPrompt.event[#p.link.eventPrompt_11].trigger2;
      R "dbEVENT".eventPrompt.event[#p.link.eventPrompt_11].trigger3;
      R "dbEVENT".eventPrompt.event[#p.link.eventPrompt_11].trigger4;
      R "dbEVENT".eventPrompt.event[#p.link.eventPrompt_11].trigger5;
      S "dbEVENT".eventPrompt.event[#p.link.eventPrompt_11].cancel1;
      S "dbEVENT".eventPrompt.event[#p.link.eventPrompt_11].cancel2;
      S "dbEVENT".eventPrompt.event[#p.link.eventPrompt_11].cancel3;
      S "dbEVENT".eventPrompt.event[#p.link.eventPrompt_11].cancel4;
      S "dbEVENT".eventPrompt.event[#p.link.eventPrompt_11].cancel5;
_not_eventPrompt_41_response:      NOP 0;

      O "dbEVENT".eventPrompt.event[#p.link.eventPrompt_12].confirmYes;
      O "dbEVENT".eventPrompt.event[#p.link.eventPrompt_12].confirmNo;
      JCN _not_eventPrompt_42_response;
      R "dbEVENT".eventPrompt.event[#p.link.eventPrompt_12].trigger1;
      R "dbEVENT".eventPrompt.event[#p.link.eventPrompt_12].trigger2;
      R "dbEVENT".eventPrompt.event[#p.link.eventPrompt_12].trigger3;
      R "dbEVENT".eventPrompt.event[#p.link.eventPrompt_12].trigger4;
      R "dbEVENT".eventPrompt.event[#p.link.eventPrompt_12].trigger5;
      S "dbEVENT".eventPrompt.event[#p.link.eventPrompt_12].cancel1;
      S "dbEVENT".eventPrompt.event[#p.link.eventPrompt_12].cancel2;
      S "dbEVENT".eventPrompt.event[#p.link.eventPrompt_12].cancel3;
      S "dbEVENT".eventPrompt.event[#p.link.eventPrompt_12].cancel4;
      S "dbEVENT".eventPrompt.event[#p.link.eventPrompt_12].cancel5;
_not_eventPrompt_42_response:      NOP 0;


NETWORK
TITLE = Return operator confirm bits if made
//------------------------------------------------------------------------//
// Receive the eventPrompt confirm bits from the global event datablock:  //
//------------------------------------------------------------------------//
      A "dbEVENT".eventPrompt.event[#p.link.eventPrompt_1].confirmYes;
      JCN _not_eventPrompt_31_confirmYes;
      S #UO_MX_FILL._prompt_abort_confirm_yes;
      R "dbEVENT".eventPrompt.event[#p.link.eventPrompt_1].confirmYes;
      R "dbEVENT".eventPrompt.event[#p.link.eventPrompt_1].confirmNo;
_not_eventPrompt_31_confirmYes:      NOP 0;
      A "dbEVENT".eventPrompt.event[#p.link.eventPrompt_2].confirmYes;
      JCN _not_eventPrompt_32_confirmYes;
      S #UO_MX_FILTER._prompt_abort_confirm_yes;
      R "dbEVENT".eventPrompt.event[#p.link.eventPrompt_2].confirmYes;
      R "dbEVENT".eventPrompt.event[#p.link.eventPrompt_2].confirmNo;
_not_eventPrompt_32_confirmYes:      NOP 0;
      A "dbEVENT".eventPrompt.event[#p.link.eventPrompt_3].confirmYes;
      JCN _not_eventPrompt_33_confirmYes;
      S #UO_MX_SETUP._prompt_connect_ok_confirm_yes;
      R "dbEVENT".eventPrompt.event[#p.link.eventPrompt_3].confirmYes;
      R "dbEVENT".eventPrompt.event[#p.link.eventPrompt_3].confirmNo;
_not_eventPrompt_33_confirmYes:      NOP 0;
      A "dbEVENT".eventPrompt.event[#p.link.eventPrompt_4].confirmYes;
      JCN _not_eventPrompt_34_confirmYes;
      S #UO_MX_FILTER._prompt_filt_completed_confirm_yes;
      R "dbEVENT".eventPrompt.event[#p.link.eventPrompt_4].confirmYes;
      R "dbEVENT".eventPrompt.event[#p.link.eventPrompt_4].confirmNo;
_not_eventPrompt_34_confirmYes:      NOP 0;
      A "dbEVENT".eventPrompt.event[#p.link.eventPrompt_5].confirmYes;
      JCN _not_eventPrompt_35_confirmYes;
      S #UO_MX_FILL._prompt_filtration_confirm_yes;
      R "dbEVENT".eventPrompt.event[#p.link.eventPrompt_5].confirmYes;
      R "dbEVENT".eventPrompt.event[#p.link.eventPrompt_5].confirmNo;
_not_eventPrompt_35_confirmYes:      NOP 0;
      A "dbEVENT".eventPrompt.event[#p.link.eventPrompt_6].confirmYes;
      JCN _not_eventPrompt_36_confirmYes;
      S #UO_MX_FILTER._prompt_filtration_confirm_yes;
      R "dbEVENT".eventPrompt.event[#p.link.eventPrompt_6].confirmYes;
      R "dbEVENT".eventPrompt.event[#p.link.eventPrompt_6].confirmNo;
_not_eventPrompt_36_confirmYes:      NOP 0;
      A "dbEVENT".eventPrompt.event[#p.link.eventPrompt_7].confirmYes;
      JCN _not_eventPrompt_37_confirmYes;
      S #UO_MX_MAKE._prompt_manway_complete_confirm_yes;
      R "dbEVENT".eventPrompt.event[#p.link.eventPrompt_7].confirmYes;
      R "dbEVENT".eventPrompt.event[#p.link.eventPrompt_7].confirmNo;
_not_eventPrompt_37_confirmYes:      NOP 0;
      A "dbEVENT".eventPrompt.event[#p.link.eventPrompt_8].confirmYes;
      JCN _not_eventPrompt_38_confirmYes;
      S #UO_MX_SETUP._prompt_not_held_confirm_yes;
      R "dbEVENT".eventPrompt.event[#p.link.eventPrompt_8].confirmYes;
      R "dbEVENT".eventPrompt.event[#p.link.eventPrompt_8].confirmNo;
_not_eventPrompt_38_confirmYes:      NOP 0;
      A "dbEVENT".eventPrompt.event[#p.link.eventPrompt_8].confirmNo;
      JCN _not_eventPrompt_38_confirmNo;
      S #UO_MX_SETUP._prompt_not_held_confirm_no;
      R "dbEVENT".eventPrompt.event[#p.link.eventPrompt_8].confirmNo;
      R "dbEVENT".eventPrompt.event[#p.link.eventPrompt_8].confirmYes;
_not_eventPrompt_38_confirmNo:      NOP 0;

      A "dbEVENT".eventPrompt.event[#p.link.eventPrompt_9].confirmYes;
      JCN _not_eventPrompt_39_confirmYes;
      S #UO_MX_SETUP._prompt_not_reach_confirm_yes;
      R "dbEVENT".eventPrompt.event[#p.link.eventPrompt_9].confirmYes;
      R "dbEVENT".eventPrompt.event[#p.link.eventPrompt_9].confirmNo;
_not_eventPrompt_39_confirmYes:      NOP 0;
      A "dbEVENT".eventPrompt.event[#p.link.eventPrompt_9].confirmNo;
      JCN _not_eventPrompt_39_confirmNo;
      S #UO_MX_SETUP._prompt_not_reach_confirm_no;
      R "dbEVENT".eventPrompt.event[#p.link.eventPrompt_9].confirmNo;
      R "dbEVENT".eventPrompt.event[#p.link.eventPrompt_9].confirmYes;
_not_eventPrompt_39_confirmNo:      NOP 0;

      A "dbEVENT".eventPrompt.event[#p.link.eventPrompt_10].confirmYes;
      JCN _not_eventPrompt_40_confirmYes;
      S #UO_MX_MAKE._prompt_pmo_confirm_yes;
      R "dbEVENT".eventPrompt.event[#p.link.eventPrompt_10].confirmYes;
      R "dbEVENT".eventPrompt.event[#p.link.eventPrompt_10].confirmNo;
_not_eventPrompt_40_confirmYes:      NOP 0;
      A "dbEVENT".eventPrompt.event[#p.link.eventPrompt_11].confirmYes;
      JCN _not_eventPrompt_41_confirmYes;
      S #UO_MX_MAKE._prompt_tare_confirm_yes;
      R "dbEVENT".eventPrompt.event[#p.link.eventPrompt_11].confirmYes;
      R "dbEVENT".eventPrompt.event[#p.link.eventPrompt_11].confirmNo;
_not_eventPrompt_41_confirmYes:      NOP 0;
      A "dbEVENT".eventPrompt.event[#p.link.eventPrompt_12].confirmYes;
      JCN _not_eventPrompt_42_confirmYes;
      S #UO_MX_SIP._prompt_try_again_confirm_yes;
      R "dbEVENT".eventPrompt.event[#p.link.eventPrompt_12].confirmYes;
      R "dbEVENT".eventPrompt.event[#p.link.eventPrompt_12].confirmNo;
_not_eventPrompt_42_confirmYes:      NOP 0;
      A "dbEVENT".eventPrompt.event[#p.link.eventPrompt_12].confirmNo;
      JCN _not_eventPrompt_42_confirmNo;
      S #UO_MX_SIP._prompt_try_again_confirm_no;
      R "dbEVENT".eventPrompt.event[#p.link.eventPrompt_12].confirmNo;
      R "dbEVENT".eventPrompt.event[#p.link.eventPrompt_12].confirmYes;
_not_eventPrompt_42_confirmNo:      NOP 0;


NETWORK
TITLE = Log prompt confirm No if required
//------------------------------------------------------------------------//
// LOG PROMPT CONFIRM NO   LOG PROMPT CONFIRM NO   LOG PROMPT CONFIRM NO  //
//                                                                        //
// Set the eventPrompt confirm No message alarm bit if active:            //
//------------------------------------------------------------------------//
      O #subsRunning.CIP;
      O #subsRunning.FILL;
      O #subsRunning.FILTER;
      O #subsRunning.MAKE;
      O #subsRunning.SETUP;
      O #subsRunning.SIP;
      JCN _noRunConfirmNo;
      A #UO_MX_SETUP._prompt_not_held_confirm_no;
      = #bEventConfirmNo[0];
      A #UO_MX_SETUP._prompt_not_reach_confirm_no;
      = #bEventConfirmNo[1];
      A #UO_MX_SIP._prompt_try_again_confirm_no;
      = #bEventConfirmNo[2];

_noRunConfirmNo:      NOP 0;

NETWORK
TITLE = Log prompt confirm Yes if required
//------------------------------------------------------------------------//
// LOG PROMPT CONFIRM YES   LOG PROMPT CONFIRM YES   LOG PROMPT CONFIRM   //
//                                                                        //
// Set the eventPrompt confirm Yes message alarm bit if active:           //
//------------------------------------------------------------------------//
      O #subsRunning.CIP;
      O #subsRunning.FILL;
      O #subsRunning.FILTER;
      O #subsRunning.MAKE;
      O #subsRunning.SETUP;
      O #subsRunning.SIP;
      JCN _noRunConfirmYes;
      A #UO_MX_FILL._prompt_abort_confirm_yes;
      = #bEventConfirmYes[0];
      A #UO_MX_FILTER._prompt_abort_confirm_yes;
      = #bEventConfirmYes[1];
      A #UO_MX_SETUP._prompt_connect_ok_confirm_yes;
      = #bEventConfirmYes[2];
      A #UO_MX_FILTER._prompt_filt_completed_confirm_yes;
      = #bEventConfirmYes[3];
      A #UO_MX_FILL._prompt_filtration_confirm_yes;
      = #bEventConfirmYes[4];
      A #UO_MX_FILTER._prompt_filtration_confirm_yes;
      = #bEventConfirmYes[5];
      A #UO_MX_MAKE._prompt_manway_complete_confirm_yes;
      = #bEventConfirmYes[6];
      A #UO_MX_SETUP._prompt_not_held_confirm_yes;
      = #bEventConfirmYes[7];
      A #UO_MX_SETUP._prompt_not_reach_confirm_yes;
      = #bEventConfirmYes[8];
      A #UO_MX_MAKE._prompt_pmo_confirm_yes;
      = #bEventConfirmYes[9];
      A #UO_MX_MAKE._prompt_tare_confirm_yes;
      = #bEventConfirmYes[10];
      A #UO_MX_SIP._prompt_try_again_confirm_yes;
      = #bEventConfirmYes[11];

_noRunConfirmYes:      NOP 0;

NETWORK
TITLE = Log message if required
//------------------------------------------------------------------------//
// LOG MSG   LOG MSG   LOG MSG   LOG MSG   LOG MSG   LOG MSG   LOG MSG    //
//                                                                        //
// Set the eventLogMsg message alarm bit if active:                       //
//------------------------------------------------------------------------//
      O #subsRunning.CIP;
      O #subsRunning.FILL;
      O #subsRunning.FILTER;
      O #subsRunning.MAKE;
      O #subsRunning.SETUP;
      O #subsRunning.SIP;
      JCN _noRunLogMsg;
      A #UO_MX_CIP._log_msg_cip_begin ;// Bit 0
      = #bEventLogMsg[0];
      R #UO_MX_CIP._log_msg_cip_begin;

      A #UO_MX_CIP._log_msg_cip_end ;// Bit 1
      = #bEventLogMsg[1];
      R #UO_MX_CIP._log_msg_cip_end;

      A #UO_MX_FILL._log_msg_fill_begin ;// Bit 2
      = #bEventLogMsg[2];
      R #UO_MX_FILL._log_msg_fill_begin;

      A #UO_MX_FILL._log_msg_fill_end ;// Bit 3
      = #bEventLogMsg[3];
      R #UO_MX_FILL._log_msg_fill_end;

      A #UO_MX_FILTER._log_msg_filter_begin ;// Bit 4
      = #bEventLogMsg[4];
      R #UO_MX_FILTER._log_msg_filter_begin;

      A #UO_MX_FILTER._log_msg_filter_end ;// Bit 5
      = #bEventLogMsg[5];
      R #UO_MX_FILTER._log_msg_filter_end;

      A #UO_MX_FILL._log_msg_filtration_complete ;// Bit 6
      = #bEventLogMsg[6];
      R #UO_MX_FILL._log_msg_filtration_complete;

      A #UO_MX_FILTER._log_msg_filtration_complete ;// Bit 7
      = #bEventLogMsg[7];
      R #UO_MX_FILTER._log_msg_filtration_complete;

      A #UO_MX_FILL._log_msg_filtration_end ;// Bit 8
      = #bEventLogMsg[8];
      R #UO_MX_FILL._log_msg_filtration_end;

      A #UO_MX_FILTER._log_msg_filtration_end ;// Bit 9
      = #bEventLogMsg[9];
      R #UO_MX_FILTER._log_msg_filtration_end;

      A #UO_MX_FILL._log_msg_filtration_start ;// Bit 10
      = #bEventLogMsg[10];
      R #UO_MX_FILL._log_msg_filtration_start;

      A #UO_MX_MAKE._log_msg_make_begin ;// Bit 11
      = #bEventLogMsg[11];
      R #UO_MX_MAKE._log_msg_make_begin;

      A #UO_MX_MAKE._log_msg_make_end ;// Bit 12
      = #bEventLogMsg[12];
      R #UO_MX_MAKE._log_msg_make_end;

      A #UO_MX_SETUP._log_msg_not_held_abort ;// Bit 13
      = #bEventLogMsg[13];
      R #UO_MX_SETUP._log_msg_not_held_abort;

      A #UO_MX_SETUP._log_msg_not_held_repeat ;// Bit 14
      = #bEventLogMsg[14];
      R #UO_MX_SETUP._log_msg_not_held_repeat;

      A #UO_MX_SETUP._log_msg_not_reach_abort ;// Bit 15
      = #bEventLogMsg[15];
      R #UO_MX_SETUP._log_msg_not_reach_abort;

      A #UO_MX_SETUP._log_msg_not_reach_repeat ;// Bit 0
      = #bEventLogMsg[16];
      R #UO_MX_SETUP._log_msg_not_reach_repeat;

      A #UO_MX_MAKE._log_msg_pmo_complete ;// Bit 1
      = #bEventLogMsg[17];
      R #UO_MX_MAKE._log_msg_pmo_complete;

      A #UO_MX_SIP._log_msg_pres_blow_reached ;// Bit 2
      = #bEventLogMsg[18];
      R #UO_MX_SIP._log_msg_pres_blow_reached;

      A #UO_MX_SIP._log_msg_pres_leave_reached ;// Bit 3
      = #bEventLogMsg[19];
      R #UO_MX_SIP._log_msg_pres_leave_reached;

      A #UO_MX_CIP._log_msg_pw_fl_wash_begin ;// Bit 4
      = #bEventLogMsg[20];
      R #UO_MX_CIP._log_msg_pw_fl_wash_begin;

      A #UO_MX_CIP._log_msg_pw_fl_wash_end ;// Bit 5
      = #bEventLogMsg[21];
      R #UO_MX_CIP._log_msg_pw_fl_wash_end;

      A #UO_MX_CIP._log_msg_pw_flood_begin ;// Bit 6
      = #bEventLogMsg[22];
      R #UO_MX_CIP._log_msg_pw_flood_begin;

      A #UO_MX_CIP._log_msg_pw_flood_end ;// Bit 7
      = #bEventLogMsg[23];
      R #UO_MX_CIP._log_msg_pw_flood_end;

      A #UO_MX_CIP._log_msg_pw_flood_timeout ;// Bit 8
      = #bEventLogMsg[24];
      R #UO_MX_CIP._log_msg_pw_flood_timeout;

      A #UO_MX_CIP._log_msg_pw_flush_begin ;// Bit 9
      = #bEventLogMsg[25];
      R #UO_MX_CIP._log_msg_pw_flush_begin;

      A #UO_MX_CIP._log_msg_pw_flush_end ;// Bit 10
      = #bEventLogMsg[26];
      R #UO_MX_CIP._log_msg_pw_flush_end;

      A #UO_MX_CIP._log_msg_pw_wash_begin ;// Bit 11
      = #bEventLogMsg[27];
      R #UO_MX_CIP._log_msg_pw_wash_begin;

      A #UO_MX_CIP._log_msg_pw_wash_end ;// Bit 12
      = #bEventLogMsg[28];
      R #UO_MX_CIP._log_msg_pw_wash_end;

      A #UO_MX_SETUP._log_msg_setup_begin ;// Bit 13
      = #bEventLogMsg[29];
      R #UO_MX_SETUP._log_msg_setup_begin;

      A #UO_MX_SETUP._log_msg_setup_end ;// Bit 14
      = #bEventLogMsg[30];
      R #UO_MX_SETUP._log_msg_setup_end;

      A #UO_MX_SIP._log_msg_sip_abort ;// Bit 15
      = #bEventLogMsg[31];
      R #UO_MX_SIP._log_msg_sip_abort;

      A #UO_MX_SIP._log_msg_sip_begin ;// Bit 0
      = #bEventLogMsg[32];
      R #UO_MX_SIP._log_msg_sip_begin;

      A #UO_MX_SIP._log_msg_sip_complete ;// Bit 1
      = #bEventLogMsg[33];
      R #UO_MX_SIP._log_msg_sip_complete;

      A #UO_MX_SIP._log_msg_sip_end ;// Bit 2
      = #bEventLogMsg[34];
      R #UO_MX_SIP._log_msg_sip_end;

      A #UO_MX_SIP._log_msg_sip_start ;// Bit 3
      = #bEventLogMsg[35];
      R #UO_MX_SIP._log_msg_sip_start;

      A #UO_MX_SIP._log_msg_sip_timer_reset ;// Bit 4
      = #bEventLogMsg[36];
      R #UO_MX_SIP._log_msg_sip_timer_reset;

      A #UO_MX_SIP._log_msg_steam_closed ;// Bit 5
      = #bEventLogMsg[37];
      R #UO_MX_SIP._log_msg_steam_closed;

      A #UO_MX_SIP._log_msg_steam_open ;// Bit 6
      = #bEventLogMsg[38];
      R #UO_MX_SIP._log_msg_steam_open;

      A #UO_MX_FILTER._log_msg_temperature_abort ;// Bit 7
      = #bEventLogMsg[39];
      R #UO_MX_FILTER._log_msg_temperature_abort;

      A #UO_MX_SETUP._log_msg_vacuum_begin ;// Bit 8
      = #bEventLogMsg[40];
      R #UO_MX_SETUP._log_msg_vacuum_begin;

      A #UO_MX_SIP._log_msg_vacuum_begin ;// Bit 9
      = #bEventLogMsg[41];
      R #UO_MX_SIP._log_msg_vacuum_begin;

      A #UO_MX_SIP._log_msg_vacuum_fail ;// Bit 10
      = #bEventLogMsg[42];
      R #UO_MX_SIP._log_msg_vacuum_fail;

      A #UO_MX_SIP._log_msg_vacuum_fail_abort ;// Bit 11
      = #bEventLogMsg[43];
      R #UO_MX_SIP._log_msg_vacuum_fail_abort;

      A #UO_MX_SIP._log_msg_vacuum_fail_repeat ;// Bit 12
      = #bEventLogMsg[44];
      R #UO_MX_SIP._log_msg_vacuum_fail_repeat;

      A #UO_MX_CIP._log_msg_wfi_rinse_begin ;// Bit 13
      = #bEventLogMsg[45];
      R #UO_MX_CIP._log_msg_wfi_rinse_begin;

      A #UO_MX_CIP._log_msg_wfi_rinse_end ;// Bit 14
      = #bEventLogMsg[46];
      R #UO_MX_CIP._log_msg_wfi_rinse_end;

      A #UO_MX_FILL._log_msg_wrong_hygiene ;// Bit 15
      = #bEventLogMsg[47];
      R #UO_MX_FILL._log_msg_wrong_hygiene;

      A #UO_MX_FILTER._log_msg_wrong_hygiene ;// Bit 0
      = #bEventLogMsg[48];
      R #UO_MX_FILTER._log_msg_wrong_hygiene;


_noRunLogMsg:      NOP 0;

NETWORK
TITLE = Real data
//------------------------------------------------------------------------//
// REAL DATA   REAL DATA   REAL DATA   REAL DATA   REAL DATA   REAL DATA  //
//                                                                        //
// Transfer the SFC eventLogReal real data to the global event datablock: //
//------------------------------------------------------------------------//
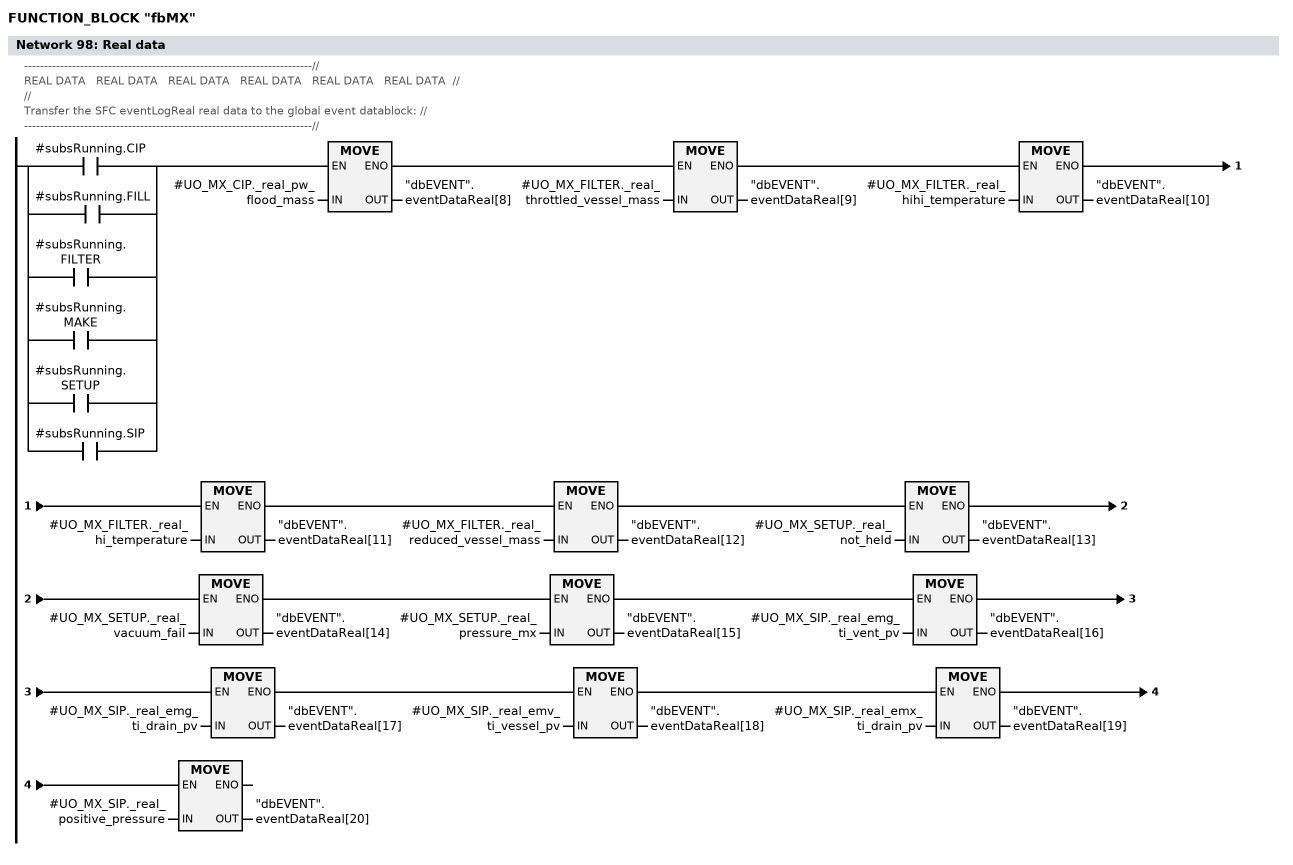
      O #subsRunning.CIP;
      O #subsRunning.FILL;
      O #subsRunning.FILTER;
      O #subsRunning.MAKE;
      O #subsRunning.SETUP;
      O #subsRunning.SIP;
      JCN _noRunLogReal;
      L #UO_MX_CIP._real_pw_flood_mass;
      T "dbEVENT".eventDataReal[8];
      L #UO_MX_FILTER._real_throttled_vessel_mass;
      T "dbEVENT".eventDataReal[9];
      L #UO_MX_FILTER._real_hihi_temperature;
      T "dbEVENT".eventDataReal[10];
      L #UO_MX_FILTER._real_hi_temperature;
      T "dbEVENT".eventDataReal[11];
      L #UO_MX_FILTER._real_reduced_vessel_mass;
      T "dbEVENT".eventDataReal[12];
      L #UO_MX_SETUP._real_not_held;
      T "dbEVENT".eventDataReal[13];
      L #UO_MX_SETUP._real_vacuum_fail;
      T "dbEVENT".eventDataReal[14];
      L #UO_MX_SETUP._real_pressure_mx;
      T "dbEVENT".eventDataReal[15];
      L #UO_MX_SIP._real_emg_ti_vent_pv;
      T "dbEVENT".eventDataReal[16];
      L #UO_MX_SIP._real_emg_ti_drain_pv;
      T "dbEVENT".eventDataReal[17];
      L #UO_MX_SIP._real_emv_ti_vessel_pv;
      T "dbEVENT".eventDataReal[18];
      L #UO_MX_SIP._real_emx_ti_drain_pv;
      T "dbEVENT".eventDataReal[19];
      L #UO_MX_SIP._real_positive_pressure;
      T "dbEVENT".eventDataReal[20];
_noRunLogReal:      NOP 0;

NETWORK
TITLE = Log real data if required
//------------------------------------------------------------------------//
// LOG REAL   LOG REAL   LOG REAL   LOG REAL   LOG REAL   LOG REAL   LOG  //
//                                                                        //
// Set the eventLogReal data alarm bit if active:                         //
//------------------------------------------------------------------------//
      O #subsRunning.CIP;
      O #subsRunning.FILL;
      O #subsRunning.FILTER;
      O #subsRunning.MAKE;
      O #subsRunning.SETUP;
      O #subsRunning.SIP;
      JCN _noRunLogRealData;
      A #UO_MX_SIP._log_real_emg_ti_drain_pv ;// Bit 0
      = #bEventLogReal[0];
      R #UO_MX_SIP._log_real_emg_ti_drain_pv;

      A #UO_MX_SIP._log_real_emg_ti_vent_pv ;// Bit 1
      = #bEventLogReal[1];
      R #UO_MX_SIP._log_real_emg_ti_vent_pv;

      A #UO_MX_SIP._log_real_emv_ti_vessel_pv ;// Bit 2
      = #bEventLogReal[2];
      R #UO_MX_SIP._log_real_emv_ti_vessel_pv;

      A #UO_MX_SIP._log_real_emx_ti_drain_pv ;// Bit 3
      = #bEventLogReal[3];
      R #UO_MX_SIP._log_real_emx_ti_drain_pv;

      A #UO_MX_FILTER._log_real_hi_temperature ;// Bit 4
      = #bEventLogReal[4];
      R #UO_MX_FILTER._log_real_hi_temperature;

      A #UO_MX_FILTER._log_real_hihi_temperature ;// Bit 5
      = #bEventLogReal[5];
      R #UO_MX_FILTER._log_real_hihi_temperature;

      A #UO_MX_SETUP._log_real_not_held ;// Bit 6
      = #bEventLogReal[6];
      R #UO_MX_SETUP._log_real_not_held;

      A #UO_MX_SIP._log_real_positive_pressure ;// Bit 7
      = #bEventLogReal[7];
      R #UO_MX_SIP._log_real_positive_pressure;

      A #UO_MX_SETUP._log_real_pressure_mx ;// Bit 8
      = #bEventLogReal[8];
      R #UO_MX_SETUP._log_real_pressure_mx;

      A #UO_MX_CIP._log_real_pw_flood_mass ;// Bit 9
      = #bEventLogReal[9];
      R #UO_MX_CIP._log_real_pw_flood_mass;

      A #UO_MX_FILTER._log_real_reduced_vessel_mass ;// Bit 10
      = #bEventLogReal[10];
      R #UO_MX_FILTER._log_real_reduced_vessel_mass;

      A #UO_MX_FILTER._log_real_throttled_vessel_mass ;// Bit 11
      = #bEventLogReal[11];
      R #UO_MX_FILTER._log_real_throttled_vessel_mass;

      A #UO_MX_SETUP._log_real_vacuum_fail ;// Bit 12
      = #bEventLogReal[12];
      R #UO_MX_SETUP._log_real_vacuum_fail;


_noRunLogRealData:      NOP 0;

NETWORK
TITLE = Time data
//------------------------------------------------------------------------//
// TIME DATA   TIME DATA   TIME DATA   TIME DATA   TIME DATA   TIME DATA  //
//                                                                        //
// Transfer the SFC eventLogTime data to the global event datablock:      //
//------------------------------------------------------------------------//
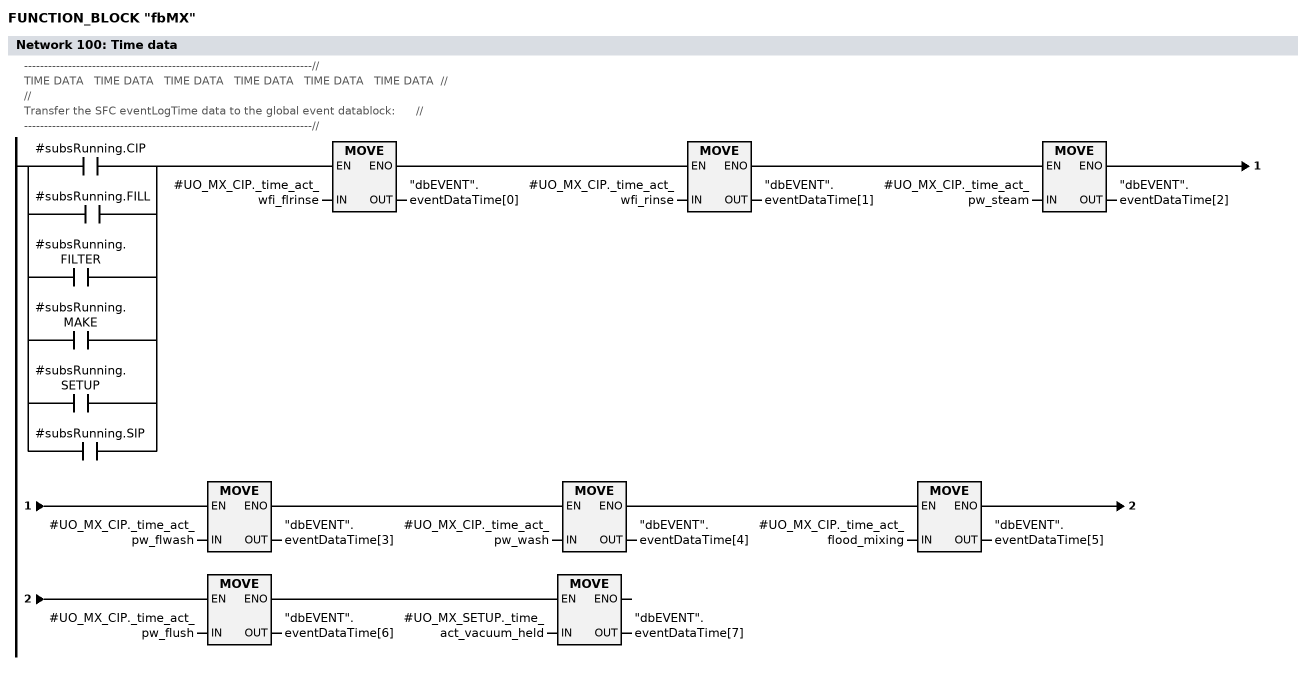
      O #subsRunning.CIP;
      O #subsRunning.FILL;
      O #subsRunning.FILTER;
      O #subsRunning.MAKE;
      O #subsRunning.SETUP;
      O #subsRunning.SIP;
      JCN _noRunLogTime;
      L #UO_MX_CIP._time_act_wfi_flrinse;
      T "dbEVENT".eventDataTime[0];
      L #UO_MX_CIP._time_act_wfi_rinse;
      T "dbEVENT".eventDataTime[1];
      L #UO_MX_CIP._time_act_pw_steam;
      T "dbEVENT".eventDataTime[2];
      L #UO_MX_CIP._time_act_pw_flwash;
      T "dbEVENT".eventDataTime[3];
      L #UO_MX_CIP._time_act_pw_wash;
      T "dbEVENT".eventDataTime[4];
      L #UO_MX_CIP._time_act_flood_mixing;
      T "dbEVENT".eventDataTime[5];
      L #UO_MX_CIP._time_act_pw_flush;
      T "dbEVENT".eventDataTime[6];
      L #UO_MX_SETUP._time_act_vacuum_held;
      T "dbEVENT".eventDataTime[7];
_noRunLogTime:      NOP 0;

NETWORK
TITLE = Log time data if required
//------------------------------------------------------------------------//
// LOG TIME   LOG TIME   LOG TIME   LOG TIME   LOG TIME   LOG TIME   LOG  //
//                                                                        //
// Set the eventLogTime data alarm bit if active:                         //
//------------------------------------------------------------------------//
      O #subsRunning.CIP;
      O #subsRunning.FILL;
      O #subsRunning.FILTER;
      O #subsRunning.MAKE;
      O #subsRunning.SETUP;
      O #subsRunning.SIP;
      JCN _noRunLogTimeData;
      A #UO_MX_CIP._log_time_act_flood_mixing ;// Bit 0
      = #bEventLogTime[0];
      R #UO_MX_CIP._log_time_act_flood_mixing;
_not_UO_MX_CIP_log_time_act_flood_mixing:      NOP 0;

      A #UO_MX_CIP._log_time_act_pw_flush ;// Bit 1
      = #bEventLogTime[1];
      R #UO_MX_CIP._log_time_act_pw_flush;
_not_UO_MX_CIP_log_time_act_pw_flush:      NOP 0;

      A #UO_MX_CIP._log_time_act_pw_flwash ;// Bit 2
      = #bEventLogTime[2];
      R #UO_MX_CIP._log_time_act_pw_flwash;
_not_UO_MX_CIP_log_time_act_pw_flwash:      NOP 0;

      A #UO_MX_CIP._log_time_act_pw_steam ;// Bit 3
      = #bEventLogTime[3];
      R #UO_MX_CIP._log_time_act_pw_steam;
_not_UO_MX_CIP_log_time_act_pw_steam:      NOP 0;

      A #UO_MX_CIP._log_time_act_pw_wash ;// Bit 4
      = #bEventLogTime[4];
      R #UO_MX_CIP._log_time_act_pw_wash;
_not_UO_MX_CIP_log_time_act_pw_wash:      NOP 0;

      A #UO_MX_SETUP._log_time_act_vacuum_held ;// Bit 5
      = #bEventLogTime[5];
      R #UO_MX_SETUP._log_time_act_vacuum_held;
_not_UO_MX_SETUP_log_time_act_vacuum_held:      NOP 0;

      A #UO_MX_CIP._log_time_act_wfi_flrinse ;// Bit 6
      = #bEventLogTime[6];
      R #UO_MX_CIP._log_time_act_wfi_flrinse;
_not_UO_MX_CIP_log_time_act_wfi_flrinse:      NOP 0;

      A #UO_MX_CIP._log_time_act_wfi_rinse ;// Bit 7
      = #bEventLogTime[7];
      R #UO_MX_CIP._log_time_act_wfi_rinse;
_not_UO_MX_CIP_log_time_act_wfi_rinse:      NOP 0;


_noRunLogTimeData:      NOP 0;

NETWORK
TITLE = Flag SFC finished if successfully completed execution
//------------------------------------------------------------------------//
// SFC COMPLETE   SFC COMPLETE   SFC COMPLETE   SFC COMPLETE   SFC COMPL  //
//                                                                        //
// Flag SFC completed if the sequence has finished executing:             //
//------------------------------------------------------------------------//
      O(;
      A #subsRunning.CIP;
      A(;
      L #UO_MX_CIP.smc.SQ_STATE;
      L "dbCONST".SEQ.STATE.COMPLETED;
      ==I;
      );
      );
      O(;
      A #subsRunning.FILL;
      A(;
      L #UO_MX_FILL.smc.SQ_STATE;
      L "dbCONST".SEQ.STATE.COMPLETED;
      ==I;
      );
      );
      O(;
      A #subsRunning.FILTER;
      A(;
      L #UO_MX_FILTER.smc.SQ_STATE;
      L "dbCONST".SEQ.STATE.COMPLETED;
      ==I;
      );
      );
      O(;
      A #subsRunning.MAKE;
      A(;
      L #UO_MX_MAKE.smc.SQ_STATE;
      L "dbCONST".SEQ.STATE.COMPLETED;
      ==I;
      );
      );
      O(;
      A #subsRunning.SETUP;
      A(;
      L #UO_MX_SETUP.smc.SQ_STATE;
      L "dbCONST".SEQ.STATE.COMPLETED;
      ==I;
      );
      );
      O(;
      A #subsRunning.SIP;
      A(;
      L #UO_MX_SIP.smc.SQ_STATE;
      L "dbCONST".SEQ.STATE.COMPLETED;
      ==I;
      );
      );
      JCN _notFinishedSuccessful;
      S #flags.sfcCompleted;
_notFinishedSuccessful:      NOP 0;

NETWORK
TITLE = Flag SFC aborted if unsuccessfully completed execution
//------------------------------------------------------------------------//
// Flag SFC completed if the sequence has been aborted:                   //
//------------------------------------------------------------------------//
      O(;
      A #subsRunning.CIP;
      A(;
      O(;
      L #UO_MX_CIP.smc.SQ_STATE;
      L "dbCONST".SEQ.STATE.ABORTED;
      ==I;
      );
      O(;
      L "dbCONST".SEQ.STATE.OFF_IDLE;
      L #UO_MX_CIP.smc.SQ_STATE;
      ==I;
      );
      );
      );
      O(;
      A #subsRunning.FILL;
      A(;
      O(;
      L #UO_MX_FILL.smc.SQ_STATE;
      L "dbCONST".SEQ.STATE.ABORTED;
      ==I;
      );
      O(;
      L "dbCONST".SEQ.STATE.OFF_IDLE;
      L #UO_MX_FILL.smc.SQ_STATE;
      ==I;
      );
      );
      );
      O(;
      A #subsRunning.FILTER;
      A(;
      O(;
      L #UO_MX_FILTER.smc.SQ_STATE;
      L "dbCONST".SEQ.STATE.ABORTED;
      ==I;
      );
      O(;
      L "dbCONST".SEQ.STATE.OFF_IDLE;
      L #UO_MX_FILTER.smc.SQ_STATE;
      ==I;
      );
      );
      );
      O(;
      A #subsRunning.MAKE;
      A(;
      O(;
      L #UO_MX_MAKE.smc.SQ_STATE;
      L "dbCONST".SEQ.STATE.ABORTED;
      ==I;
      );
      O(;
      L "dbCONST".SEQ.STATE.OFF_IDLE;
      L #UO_MX_MAKE.smc.SQ_STATE;
      ==I;
      );
      );
      );
      O(;
      A #subsRunning.SETUP;
      A(;
      O(;
      L #UO_MX_SETUP.smc.SQ_STATE;
      L "dbCONST".SEQ.STATE.ABORTED;
      ==I;
      );
      O(;
      L "dbCONST".SEQ.STATE.OFF_IDLE;
      L #UO_MX_SETUP.smc.SQ_STATE;
      ==I;
      );
      );
      );
      O(;
      A #subsRunning.SIP;
      A(;
      O(;
      L #UO_MX_SIP.smc.SQ_STATE;
      L "dbCONST".SEQ.STATE.ABORTED;
      ==I;
      );
      O(;
      L "dbCONST".SEQ.STATE.OFF_IDLE;
      L #UO_MX_SIP.smc.SQ_STATE;
      ==I;
      );
      );
      );
      JCN _notFinishedUnsuccessful;
      S #flags.sfcAborted;
      S #flags.substateCompleted;
      L "dbCONST".BLK.MX.STATE.ABORTED;
      T #p.read.mc.STATE;
_notFinishedUnsuccessful:      NOP 0;

NETWORK
TITLE = Check if substate completed
//------------------------------------------------------------------------//
// Check if substate has been completed if SFC finished if there is one:  //
//------------------------------------------------------------------------//
      O(;
      A #subsRunning.CIP;
      A(;
      O(;
      A #subsHasSFC.CIP;
      A #flags.sfcCompleted;
      );
      ON #subsHasSFC.CIP;
      );
      );
      O(;
      A #subsRunning.FILL;
      A(;
      O(;
      A #subsHasSFC.FILL;
      A #flags.sfcCompleted;
      );
      ON #subsHasSFC.FILL;
      );
      );
      O(;
      A #subsRunning.FILTER;
      A(;
      O(;
      A #subsHasSFC.FILTER;
      A #flags.sfcCompleted;
      );
      ON #subsHasSFC.FILTER;
      );
      );
      O(;
      A #subsRunning.MAKE;
      A(;
      O(;
      A #subsHasSFC.MAKE;
      A #flags.sfcCompleted;
      );
      ON #subsHasSFC.MAKE;
      );
      );
      O(;
      A #subsRunning.SETUP;
      A(;
      O(;
      A #subsHasSFC.SETUP;
      A #flags.sfcCompleted;
      );
      ON #subsHasSFC.SETUP;
      );
      );
      O(;
      A #subsRunning.SIP;
      A(;
      O(;
      A #subsHasSFC.SIP;
      A #flags.sfcCompleted;
      );
      ON #subsHasSFC.SIP;
      );
      );
      JCN _noSubstateComplete;
      S #flags.substateCompleted;
_noSubstateComplete:      NOP 0;

      SET;
      JC _switch_end;

  //------------------------------------------------------------------------//
  // SWITCH   SWITCH   SWITCH   SWITCH   SWITCH   SWITCH   SWITCH   SWITCH  //
  // COMPLETED   COMPLETED   COMPLETED   COMPLETED   COMPLETED   COMPLETED  //
  // COMPLETED   COMPLETED   COMPLETED   COMPLETED   COMPLETED   COMPLETED  //
  //------------------------------------------------------------------------//
_state_COMPLETED:      NOP 0;

NETWORK
TITLE = COMPLETED COMPLETED COMPLETED Running substate completed
//------------------------------------------------------------------------//
// BLOCK COMPLETE   BLOCK COMPLETE   BLOCK COMPLETE   BLOCK COMPLETE   BL //
//                                                                        //
// Set the block state to COMPLETED if no SFC or SFC completed:           //
//------------------------------------------------------------------------//
      AN #flags.childMismatch;
      AN #flags.sfcAborted;
      JCN _blkComplete;
      L "dbCONST".BLK.MX.STATE.COMPLETED;
      T #p.read.mc.STATE;
      L #p.write.mc.SUBS;
      T #p.read.bmc.lastSUBS;

_blkComplete:      NOP 0;

NETWORK
TITLE = Release child EMX_FILL1 if acquired and command completed
//------------------------------------------------------------------------//
// RELEASE CHILD   RELEASE CHILD   RELEASE CHILD   RELEASE CHILD   RELE   //
//                                                                        //
// Release the child device if acquired earlier to run the command:       //
//------------------------------------------------------------------------//
      A #acquire.EMX_FILL1;
      JCN _notOwn1;
      L "dbCONST".BLK.ID.AVAILABLE;
      T "idbEMX5".f[#p.child.EMX_FILL1].p.write.mc.OWNER;
      R #acquire.EMX_FILL1;
_notOwn1:      NOP 0;

NETWORK
TITLE = Release child EMX_FILL2 if acquired and command completed
//------------------------------------------------------------------------//
// RELEASE CHILD   RELEASE CHILD   RELEASE CHILD   RELEASE CHILD   RELE   //
//                                                                        //
// Release the child device if acquired earlier to run the command:       //
//------------------------------------------------------------------------//
      A #acquire.EMX_FILL2;
      JCN _notOwn2;
      L "dbCONST".BLK.ID.AVAILABLE;
      T "idbEMX5".f[#p.child.EMX_FILL2].p.write.mc.OWNER;
      R #acquire.EMX_FILL2;
_notOwn2:      NOP 0;

NETWORK
TITLE = Release child EMX_SMFL if acquired and command completed
//------------------------------------------------------------------------//
// RELEASE CHILD   RELEASE CHILD   RELEASE CHILD   RELEASE CHILD   RELE   //
//                                                                        //
// Release the child device if acquired earlier to run the command:       //
//------------------------------------------------------------------------//
      A #acquire.EMX_SMFL;
      JCN _notOwn3;
      L "dbCONST".BLK.ID.AVAILABLE;
      T "idbEMX6".f[#p.child.EMX_SMFL].p.write.mc.OWNER;
      R #acquire.EMX_SMFL;
_notOwn3:      NOP 0;

NETWORK
TITLE = Release child EMX_SMFLDRN if acquired and command completed
//------------------------------------------------------------------------//
// RELEASE CHILD   RELEASE CHILD   RELEASE CHILD   RELEASE CHILD   RELE   //
//                                                                        //
// Release the child device if acquired earlier to run the command:       //
//------------------------------------------------------------------------//
      A #acquire.EMX_SMFLDRN;
      JCN _notOwn4;
      L "dbCONST".BLK.ID.AVAILABLE;
      T "idbEMX4".f[#p.child.EMX_SMFLDRN].p.write.mc.OWNER;
      R #acquire.EMX_SMFLDRN;
_notOwn4:      NOP 0;

NETWORK
TITLE = Release child EMX_TRANSFER1 if acquired and command completed
//------------------------------------------------------------------------//
// RELEASE CHILD   RELEASE CHILD   RELEASE CHILD   RELEASE CHILD   RELE   //
//                                                                        //
// Release the child device if acquired earlier to run the command:       //
//------------------------------------------------------------------------//
      A #acquire.EMX_TRANSFER1;
      JCN _notOwn5;
      L "dbCONST".BLK.ID.AVAILABLE;
      T "idbEMX2".f[#p.child.EMX_TRANSFER1].p.write.mc.OWNER;
      R #acquire.EMX_TRANSFER1;
_notOwn5:      NOP 0;

NETWORK
TITLE = Release child EMX_TRANSFER2 if acquired and command completed
//------------------------------------------------------------------------//
// RELEASE CHILD   RELEASE CHILD   RELEASE CHILD   RELEASE CHILD   RELE   //
//                                                                        //
// Release the child device if acquired earlier to run the command:       //
//------------------------------------------------------------------------//
      A #acquire.EMX_TRANSFER2;
      JCN _notOwn6;
      L "dbCONST".BLK.ID.AVAILABLE;
      T "idbEMX2".f[#p.child.EMX_TRANSFER2].p.write.mc.OWNER;
      R #acquire.EMX_TRANSFER2;
_notOwn6:      NOP 0;


  //------------------------------------------------------------------------//
  // SWITCH   SWITCH   SWITCH   SWITCH   SWITCH   SWITCH   SWITCH   SWITCH  //
  // END   END   END   END   END   END  END   END   END   END   END   END   //
  // END   END   END   END   END   END  END   END   END   END   END   END   //
  //------------------------------------------------------------------------//
_switch_end:      NOP 0;

NETWORK
TITLE = SWITCH END SWITCH END ERROR if child mismatch
//------------------------------------------------------------------------//
// BLOCK ERROR   BLOCK ERROR   BLOCK ERROR   BLOCK ERROR   BLOCK ERROR    //
//                                                                        //
// Set the block state to ERROR if child mismatch and not STOPPED:        //
//------------------------------------------------------------------------//
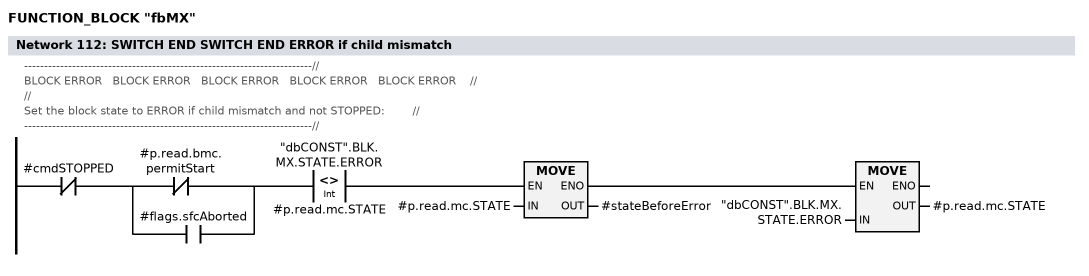
      AN #cmdSTOPPED;
      A(;
      ON #p.read.bmc.permitStart;
      O #flags.sfcAborted;
      );
      A(;
      L "dbCONST".BLK.MX.STATE.ERROR;
      L #p.read.mc.STATE;
      <>I;
      );
      JCN _blkError;
      L #p.read.mc.STATE;
      T #stateBeforeError;
      L "dbCONST".BLK.MX.STATE.ERROR;
      T #p.read.mc.STATE;
_blkError:      NOP 0;

NETWORK
TITLE = RESUME if children now okay
//------------------------------------------------------------------------//
// BLOCK RESUME   BLOCK RESUME   BLOCK RESUME   BLOCK RESUME   BLOCK RES  //
//                                                                        //
// Resume the running SFC sequence if no interlock or failure condition:  //
//------------------------------------------------------------------------//
      AN #cmdSTOPPED;
      A #p.read.bmc.permitStart;
      AN #flags.sfcAborted;
      A(;
      L "dbCONST".BLK.MX.STATE.ERROR;
      L #p.read.mc.STATE;
      ==I;
      );
      JCN _noResume;
      L #stateBeforeError;
      T #p.read.mc.STATE;

      A #subsRunning.CIP;
      JCN _resumeSFC_1;
      L "dbCONST".SEQ.CMD.RESUME;
      T #UO_MX_CIP.smc.SQ_CMD;
_resumeSFC_1:      NOP 0;

      A #subsRunning.FILL;
      JCN _resumeSFC_2;
      L "dbCONST".SEQ.CMD.RESUME;
      T #UO_MX_FILL.smc.SQ_CMD;
_resumeSFC_2:      NOP 0;

      A #subsRunning.FILTER;
      JCN _resumeSFC_3;
      L "dbCONST".SEQ.CMD.RESUME;
      T #UO_MX_FILTER.smc.SQ_CMD;
_resumeSFC_3:      NOP 0;

      A #subsRunning.MAKE;
      JCN _resumeSFC_4;
      L "dbCONST".SEQ.CMD.RESUME;
      T #UO_MX_MAKE.smc.SQ_CMD;
_resumeSFC_4:      NOP 0;

      A #subsRunning.SETUP;
      JCN _resumeSFC_5;
      L "dbCONST".SEQ.CMD.RESUME;
      T #UO_MX_SETUP.smc.SQ_CMD;
_resumeSFC_5:      NOP 0;

      A #subsRunning.SIP;
      JCN _resumeSFC_6;
      L "dbCONST".SEQ.CMD.RESUME;
      T #UO_MX_SIP.smc.SQ_CMD;
_resumeSFC_6:      NOP 0;


_noResume:      NOP 0;

NETWORK
TITLE = Upload child states
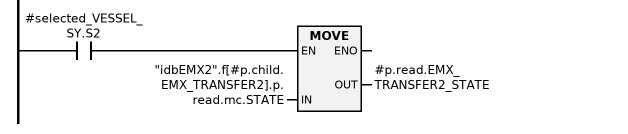
      A "alwaysHigh";
      JCN _pSTATE_DI_ASL;
      L "idbDI1".f[#p.child.DI_ASL].p.read.mc.STATE;
      T #p.read.DI_ASL_STATE;
_pSTATE_DI_ASL:      NOP 0;

      A "alwaysHigh";
      JCN _pSTATE_DI_ESTOP;
      L "idbDI1".f[#p.child.DI_ESTOP].p.read.mc.STATE;
      T #p.read.DI_ESTOP_STATE;
_pSTATE_DI_ESTOP:      NOP 0;

      A "alwaysHigh";
      JCN _pSTATE_DI_ESTOP_AUX1;
      L "idbDI1".f[#p.child.DI_ESTOP_AUX1].p.read.mc.STATE;
      T #p.read.DI_ESTOP_AUX1_STATE;
_pSTATE_DI_ESTOP_AUX1:      NOP 0;

      A "alwaysHigh";
      JCN _pSTATE_DI_ESTOP_AUX2;
      L "idbDI1".f[#p.child.DI_ESTOP_AUX2].p.read.mc.STATE;
      T #p.read.DI_ESTOP_AUX2_STATE;
_pSTATE_DI_ESTOP_AUX2:      NOP 0;

      A "alwaysHigh";
      JCN _pSTATE_DI_ESTOP_AUX3;
      L "idbDI1".f[#p.child.DI_ESTOP_AUX3].p.read.mc.STATE;
      T #p.read.DI_ESTOP_AUX3_STATE;
_pSTATE_DI_ESTOP_AUX3:      NOP 0;

      A "alwaysHigh";
      JCN _pSTATE_DI_RELAY;
      L "idbDI2".f[#p.child.DI_RELAY].p.read.mc.STATE;
      T #p.read.DI_RELAY_STATE;
_pSTATE_DI_RELAY:      NOP 0;

      A "alwaysHigh";
      JCN _pSTATE_EMA_VESSEL;
      L "idbEMA1".f[#p.child.EMA_VESSEL].p.read.mc.STATE;
      T #p.read.EMA_VESSEL_STATE;
_pSTATE_EMA_VESSEL:      NOP 0;

      A "alwaysHigh";
      JCN _pSTATE_EMC_GAS;
      L "idbEMC1".f[#p.child.EMC_GAS].p.read.mc.STATE;
      T #p.read.EMC_GAS_STATE;
_pSTATE_EMC_GAS:      NOP 0;

      A "alwaysHigh";
      JCN _pSTATE_EMC_WATER;
      L "idbEMC2".f[#p.child.EMC_WATER].p.read.mc.STATE;
      T #p.read.EMC_WATER_STATE;
_pSTATE_EMC_WATER:      NOP 0;

      A "alwaysHigh";
      JCN _pSTATE_EMG_FILTER;
      L "idbEMG1".f[#p.child.EMG_FILTER].p.read.mc.STATE;
      T #p.read.EMG_FILTER_STATE;
_pSTATE_EMG_FILTER:      NOP 0;

      A "alwaysHigh";
      JCN _pSTATE_EMM_VESSEL;
      L "idbEMM1".f[#p.child.EMM_VESSEL].p.read.mc.STATE;
      T #p.read.EMM_VESSEL_STATE;
_pSTATE_EMM_VESSEL:      NOP 0;

      A "alwaysHigh";
      JCN _pSTATE_EMT_HEX;
      L "idbEMT1".f[#p.child.EMT_HEX].p.read.mc.STATE;
      T #p.read.EMT_HEX_STATE;
_pSTATE_EMT_HEX:      NOP 0;

      A "alwaysHigh";
      JCN _pSTATE_EMV_INLET;
      L "idbEMV2".f[#p.child.EMV_INLET].p.read.mc.STATE;
      T #p.read.EMV_INLET_STATE;
_pSTATE_EMV_INLET:      NOP 0;

      A "alwaysHigh";
      JCN _pSTATE_EMV_VESSEL;
      L "idbEMV1".f[#p.child.EMV_VESSEL].p.read.mc.STATE;
      T #p.read.EMV_VESSEL_STATE;
_pSTATE_EMV_VESSEL:      NOP 0;

      A "alwaysHigh";
      JCN _pSTATE_EMX_DRAIN;
      L "idbEMX4".f[#p.child.EMX_DRAIN].p.read.mc.STATE;
      T #p.read.EMX_DRAIN_STATE;
_pSTATE_EMX_DRAIN:      NOP 0;

      A #selected_FILL_FLZ.FL1;
      JCN _pSTATE_EMX_FILL1;
      L "idbEMX5".f[#p.child.EMX_FILL1].p.read.mc.STATE;
      T #p.read.EMX_FILL1_STATE;
_pSTATE_EMX_FILL1:      NOP 0;

      A #selected_FILL_FLZ.FL2;
      JCN _pSTATE_EMX_FILL2;
      L "idbEMX5".f[#p.child.EMX_FILL2].p.read.mc.STATE;
      T #p.read.EMX_FILL2_STATE;
_pSTATE_EMX_FILL2:      NOP 0;

      A "alwaysHigh";
      JCN _pSTATE_EMX_MMFL;
      L "idbEMX1".f[#p.child.EMX_MMFL].p.read.mc.STATE;
      T #p.read.EMX_MMFL_STATE;
_pSTATE_EMX_MMFL:      NOP 0;

      O #selected_FILL_FLZ.FL1;
      O #selected_FILL_FLZ.FL2;
      O #selected_VESSEL_SY.S1;
      O #selected_VESSEL_SY.S2;
      JCN _pSTATE_EMX_SMFL;
      L "idbEMX6".f[#p.child.EMX_SMFL].p.read.mc.STATE;
      T #p.read.EMX_SMFL_STATE;
_pSTATE_EMX_SMFL:      NOP 0;

      O #selected_FILL_FLZ.FL1;
      O #selected_FILL_FLZ.FL2;
      O #selected_VESSEL_SY.S1;
      O #selected_VESSEL_SY.S2;
      JCN _pSTATE_EMX_SMFLDRN;
      L "idbEMX4".f[#p.child.EMX_SMFLDRN].p.read.mc.STATE;
      T #p.read.EMX_SMFLDRN_STATE;
_pSTATE_EMX_SMFLDRN:      NOP 0;

      A #selected_VESSEL_SY.S1;
      JCN _pSTATE_EMX_TRANSFER1;
      L "idbEMX2".f[#p.child.EMX_TRANSFER1].p.read.mc.STATE;
      T #p.read.EMX_TRANSFER1_STATE;
_pSTATE_EMX_TRANSFER1:      NOP 0;

      A #selected_VESSEL_SY.S2;
      JCN _pSTATE_EMX_TRANSFER2;
      L "idbEMX2".f[#p.child.EMX_TRANSFER2].p.read.mc.STATE;
      T #p.read.EMX_TRANSFER2_STATE;
_pSTATE_EMX_TRANSFER2:      NOP 0;



NETWORK
TITLE = Set child commands
  //------------------------------------------------------------------------//
  // Set the child substate if no child mismatch:                           //
  //------------------------------------------------------------------------//
      AN #timeCheckChildStateExpired;
      A(;
      O #p.read.bmc.stateRUNNING;
      O #flags.substateCompleted;
      );
      JCN _noCommandOnChildMismatch;

      A "idbEMA1".f[#p.child.EMA_VESSEL].p.read.mc.modeAUTO;
      A "alwaysHigh";
      JCN _pSUBS_EMA_VESSEL;
      L #p.write.EMA_VESSEL_SUBS;
      T "idbEMA1".f[#p.child.EMA_VESSEL].p.write.mc.SUBS;
_pSUBS_EMA_VESSEL:      NOP 0;

      A "idbEMC1".f[#p.child.EMC_GAS].p.read.mc.modeAUTO;
      A "alwaysHigh";
      JCN _pSUBS_EMC_GAS;
      L #p.write.EMC_GAS_SUBS;
      T "idbEMC1".f[#p.child.EMC_GAS].p.write.mc.SUBS;
_pSUBS_EMC_GAS:      NOP 0;

      A "idbEMC2".f[#p.child.EMC_WATER].p.read.mc.modeAUTO;
      A "alwaysHigh";
      JCN _pSUBS_EMC_WATER;
      L #p.write.EMC_WATER_SUBS;
      T "idbEMC2".f[#p.child.EMC_WATER].p.write.mc.SUBS;
_pSUBS_EMC_WATER:      NOP 0;

      A "idbEMG1".f[#p.child.EMG_FILTER].p.read.mc.modeAUTO;
      A "alwaysHigh";
      JCN _pSUBS_EMG_FILTER;
      L #p.write.EMG_FILTER_SUBS;
      T "idbEMG1".f[#p.child.EMG_FILTER].p.write.mc.SUBS;
_pSUBS_EMG_FILTER:      NOP 0;

      A "idbEMM1".f[#p.child.EMM_VESSEL].p.read.mc.modeAUTO;
      A "alwaysHigh";
      JCN _pSUBS_EMM_VESSEL;
      L #p.write.EMM_VESSEL_SUBS;
      T "idbEMM1".f[#p.child.EMM_VESSEL].p.write.mc.SUBS;
_pSUBS_EMM_VESSEL:      NOP 0;

      A "idbEMT1".f[#p.child.EMT_HEX].p.read.mc.modeAUTO;
      A "alwaysHigh";
      JCN _pSUBS_EMT_HEX;
      L #p.write.EMT_HEX_SUBS;
      T "idbEMT1".f[#p.child.EMT_HEX].p.write.mc.SUBS;
_pSUBS_EMT_HEX:      NOP 0;

      A "idbEMV2".f[#p.child.EMV_INLET].p.read.mc.modeAUTO;
      A "alwaysHigh";
      JCN _pSUBS_EMV_INLET;
      L #p.write.EMV_INLET_SUBS;
      T "idbEMV2".f[#p.child.EMV_INLET].p.write.mc.SUBS;
_pSUBS_EMV_INLET:      NOP 0;

      A "idbEMV1".f[#p.child.EMV_VESSEL].p.read.mc.modeAUTO;
      A "alwaysHigh";
      JCN _pSUBS_EMV_VESSEL;
      L #p.write.EMV_VESSEL_SUBS;
      T "idbEMV1".f[#p.child.EMV_VESSEL].p.write.mc.SUBS;
_pSUBS_EMV_VESSEL:      NOP 0;

      A "idbEMX4".f[#p.child.EMX_DRAIN].p.read.mc.modeAUTO;
      A "alwaysHigh";
      JCN _pSUBS_EMX_DRAIN;
      L #p.write.EMX_DRAIN_SUBS;
      T "idbEMX4".f[#p.child.EMX_DRAIN].p.write.mc.SUBS;
_pSUBS_EMX_DRAIN:      NOP 0;

      A "idbEMX5".f[#p.child.EMX_FILL1].p.read.mc.modeAUTO;
      A #selected_FILL_FLZ.FL1;
      JCN _pSUBS_EMX_FILL1;
      L #p.write.EMX_FILL1_SUBS;
      T "idbEMX5".f[#p.child.EMX_FILL1].p.write.mc.SUBS;
_pSUBS_EMX_FILL1:      NOP 0;

      A "idbEMX5".f[#p.child.EMX_FILL2].p.read.mc.modeAUTO;
      A #selected_FILL_FLZ.FL2;
      JCN _pSUBS_EMX_FILL2;
      L #p.write.EMX_FILL2_SUBS;
      T "idbEMX5".f[#p.child.EMX_FILL2].p.write.mc.SUBS;
_pSUBS_EMX_FILL2:      NOP 0;

      A "idbEMX1".f[#p.child.EMX_MMFL].p.read.mc.modeAUTO;
      A "alwaysHigh";
      JCN _pSUBS_EMX_MMFL;
      L #p.write.EMX_MMFL_SUBS;
      T "idbEMX1".f[#p.child.EMX_MMFL].p.write.mc.SUBS;
_pSUBS_EMX_MMFL:      NOP 0;

      A "idbEMX6".f[#p.child.EMX_SMFL].p.read.mc.modeAUTO;
      O #selected_FILL_FLZ.FL1;
      O #selected_FILL_FLZ.FL2;
      O #selected_VESSEL_SY.S1;
      O #selected_VESSEL_SY.S2;
      JCN _pSUBS_EMX_SMFL;
      L #p.write.EMX_SMFL_SUBS;
      T "idbEMX6".f[#p.child.EMX_SMFL].p.write.mc.SUBS;
_pSUBS_EMX_SMFL:      NOP 0;

      A "idbEMX4".f[#p.child.EMX_SMFLDRN].p.read.mc.modeAUTO;
      O #selected_FILL_FLZ.FL1;
      O #selected_FILL_FLZ.FL2;
      O #selected_VESSEL_SY.S1;
      O #selected_VESSEL_SY.S2;
      JCN _pSUBS_EMX_SMFLDRN;
      L #p.write.EMX_SMFLDRN_SUBS;
      T "idbEMX4".f[#p.child.EMX_SMFLDRN].p.write.mc.SUBS;
_pSUBS_EMX_SMFLDRN:      NOP 0;

      A "idbEMX2".f[#p.child.EMX_TRANSFER1].p.read.mc.modeAUTO;
      A #selected_VESSEL_SY.S1;
      JCN _pSUBS_EMX_TRANSFER1;
      L #p.write.EMX_TRANSFER1_SUBS;
      T "idbEMX2".f[#p.child.EMX_TRANSFER1].p.write.mc.SUBS;
_pSUBS_EMX_TRANSFER1:      NOP 0;

      A "idbEMX2".f[#p.child.EMX_TRANSFER2].p.read.mc.modeAUTO;
      A #selected_VESSEL_SY.S2;
      JCN _pSUBS_EMX_TRANSFER2;
      L #p.write.EMX_TRANSFER2_SUBS;
      T "idbEMX2".f[#p.child.EMX_TRANSFER2].p.write.mc.SUBS;
_pSUBS_EMX_TRANSFER2:      NOP 0;


  //------------------------------------------------------------------------//
  // Set the child command if no child mismatch:                            //
  //------------------------------------------------------------------------//
      A "idbEMA1".f[#p.child.EMA_VESSEL].p.read.mc.modeAUTO;
      A "alwaysHigh";
      JCN _pCMD_EMA_VESSEL;
      L #p.write.EMA_VESSEL_CMD;
      T "idbEMA1".f[#p.child.EMA_VESSEL].p.write.mc.CMD;
      T #childReqCMD.EMA_VESSEL;
_pCMD_EMA_VESSEL:      NOP 0;

      A "idbEMC1".f[#p.child.EMC_GAS].p.read.mc.modeAUTO;
      A "alwaysHigh";
      JCN _pCMD_EMC_GAS;
      L #p.write.EMC_GAS_CMD;
      T "idbEMC1".f[#p.child.EMC_GAS].p.write.mc.CMD;
      T #childReqCMD.EMC_GAS;
_pCMD_EMC_GAS:      NOP 0;

      A "idbEMC2".f[#p.child.EMC_WATER].p.read.mc.modeAUTO;
      A "alwaysHigh";
      JCN _pCMD_EMC_WATER;
      L #p.write.EMC_WATER_CMD;
      T "idbEMC2".f[#p.child.EMC_WATER].p.write.mc.CMD;
      T #childReqCMD.EMC_WATER;
_pCMD_EMC_WATER:      NOP 0;

      A "idbEMG1".f[#p.child.EMG_FILTER].p.read.mc.modeAUTO;
      A "alwaysHigh";
      JCN _pCMD_EMG_FILTER;
      L #p.write.EMG_FILTER_CMD;
      T "idbEMG1".f[#p.child.EMG_FILTER].p.write.mc.CMD;
      T #childReqCMD.EMG_FILTER;
_pCMD_EMG_FILTER:      NOP 0;

      A "idbEMM1".f[#p.child.EMM_VESSEL].p.read.mc.modeAUTO;
      A "alwaysHigh";
      JCN _pCMD_EMM_VESSEL;
      L #p.write.EMM_VESSEL_CMD;
      T "idbEMM1".f[#p.child.EMM_VESSEL].p.write.mc.CMD;
      T #childReqCMD.EMM_VESSEL;
_pCMD_EMM_VESSEL:      NOP 0;

      A "idbEMT1".f[#p.child.EMT_HEX].p.read.mc.modeAUTO;
      A "alwaysHigh";
      JCN _pCMD_EMT_HEX;
      L #p.write.EMT_HEX_CMD;
      T "idbEMT1".f[#p.child.EMT_HEX].p.write.mc.CMD;
      T #childReqCMD.EMT_HEX;
_pCMD_EMT_HEX:      NOP 0;

      A "idbEMV2".f[#p.child.EMV_INLET].p.read.mc.modeAUTO;
      A "alwaysHigh";
      JCN _pCMD_EMV_INLET;
      L #p.write.EMV_INLET_CMD;
      T "idbEMV2".f[#p.child.EMV_INLET].p.write.mc.CMD;
      T #childReqCMD.EMV_INLET;
_pCMD_EMV_INLET:      NOP 0;

      A "idbEMV1".f[#p.child.EMV_VESSEL].p.read.mc.modeAUTO;
      A "alwaysHigh";
      JCN _pCMD_EMV_VESSEL;
      L #p.write.EMV_VESSEL_CMD;
      T "idbEMV1".f[#p.child.EMV_VESSEL].p.write.mc.CMD;
      T #childReqCMD.EMV_VESSEL;
_pCMD_EMV_VESSEL:      NOP 0;

      A "idbEMX4".f[#p.child.EMX_DRAIN].p.read.mc.modeAUTO;
      A "alwaysHigh";
      JCN _pCMD_EMX_DRAIN;
      L #p.write.EMX_DRAIN_CMD;
      T "idbEMX4".f[#p.child.EMX_DRAIN].p.write.mc.CMD;
      T #childReqCMD.EMX_DRAIN;
_pCMD_EMX_DRAIN:      NOP 0;

      A "idbEMX5".f[#p.child.EMX_FILL1].p.read.mc.modeAUTO;
      A #selected_FILL_FLZ.FL1;
      JCN _pCMD_EMX_FILL1;
      L #p.write.EMX_FILL1_CMD;
      T "idbEMX5".f[#p.child.EMX_FILL1].p.write.mc.CMD;
      T #childReqCMD.EMX_FILL1;
_pCMD_EMX_FILL1:      NOP 0;

      A "idbEMX5".f[#p.child.EMX_FILL2].p.read.mc.modeAUTO;
      A #selected_FILL_FLZ.FL2;
      JCN _pCMD_EMX_FILL2;
      L #p.write.EMX_FILL2_CMD;
      T "idbEMX5".f[#p.child.EMX_FILL2].p.write.mc.CMD;
      T #childReqCMD.EMX_FILL2;
_pCMD_EMX_FILL2:      NOP 0;

      A "idbEMX1".f[#p.child.EMX_MMFL].p.read.mc.modeAUTO;
      A "alwaysHigh";
      JCN _pCMD_EMX_MMFL;
      L #p.write.EMX_MMFL_CMD;
      T "idbEMX1".f[#p.child.EMX_MMFL].p.write.mc.CMD;
      T #childReqCMD.EMX_MMFL;
_pCMD_EMX_MMFL:      NOP 0;

      A "idbEMX6".f[#p.child.EMX_SMFL].p.read.mc.modeAUTO;
      O #selected_FILL_FLZ.FL1;
      O #selected_FILL_FLZ.FL2;
      O #selected_VESSEL_SY.S1;
      O #selected_VESSEL_SY.S2;
      JCN _pCMD_EMX_SMFL;
      L #p.write.EMX_SMFL_CMD;
      T "idbEMX6".f[#p.child.EMX_SMFL].p.write.mc.CMD;
      T #childReqCMD.EMX_SMFL;
_pCMD_EMX_SMFL:      NOP 0;

      A "idbEMX4".f[#p.child.EMX_SMFLDRN].p.read.mc.modeAUTO;
      O #selected_FILL_FLZ.FL1;
      O #selected_FILL_FLZ.FL2;
      O #selected_VESSEL_SY.S1;
      O #selected_VESSEL_SY.S2;
      JCN _pCMD_EMX_SMFLDRN;
      L #p.write.EMX_SMFLDRN_CMD;
      T "idbEMX4".f[#p.child.EMX_SMFLDRN].p.write.mc.CMD;
      T #childReqCMD.EMX_SMFLDRN;
_pCMD_EMX_SMFLDRN:      NOP 0;

      A "idbEMX2".f[#p.child.EMX_TRANSFER1].p.read.mc.modeAUTO;
      A #selected_VESSEL_SY.S1;
      JCN _pCMD_EMX_TRANSFER1;
      L #p.write.EMX_TRANSFER1_CMD;
      T "idbEMX2".f[#p.child.EMX_TRANSFER1].p.write.mc.CMD;
      T #childReqCMD.EMX_TRANSFER1;
_pCMD_EMX_TRANSFER1:      NOP 0;

      A "idbEMX2".f[#p.child.EMX_TRANSFER2].p.read.mc.modeAUTO;
      A #selected_VESSEL_SY.S2;
      JCN _pCMD_EMX_TRANSFER2;
      L #p.write.EMX_TRANSFER2_CMD;
      T "idbEMX2".f[#p.child.EMX_TRANSFER2].p.write.mc.CMD;
      T #childReqCMD.EMX_TRANSFER2;
_pCMD_EMX_TRANSFER2:      NOP 0;


  //------------------------------------------------------------------------//
  // Write the non-boolean child parameters if no child mismatch:           //
  //------------------------------------------------------------------------//
      A "idbEMX4".f[#p.child.EMX_DRAIN].p.read.mc.modeAUTO;
      JCN _pSFCChildWrite_EMX_DRAIN_CLOSED_TIME;
      L #p.write.EMX_DRAIN_CLOSED_TIME;
      T "idbEMX4".f[#p.child.EMX_DRAIN].p.write.CLOSED_TIME;
_pSFCChildWrite_EMX_DRAIN_CLOSED_TIME:      NOP 0;

      A "idbEMX4".f[#p.child.EMX_DRAIN].p.read.mc.modeAUTO;
      JCN _pSFCChildWrite_EMX_DRAIN_OPENED_TIME;
      L #p.write.EMX_DRAIN_OPENED_TIME;
      T "idbEMX4".f[#p.child.EMX_DRAIN].p.write.OPENED_TIME;
_pSFCChildWrite_EMX_DRAIN_OPENED_TIME:      NOP 0;

      A "idbEMX4".f[#p.child.EMX_SMFLDRN].p.read.mc.modeAUTO;
      JCN _pSFCChildWrite_EMX_SMFLDRN_CLOSED_TIME;
      L #p.write.EMX_SMFLDRN_CLOSED_TIME;
      T "idbEMX4".f[#p.child.EMX_SMFLDRN].p.write.CLOSED_TIME;
_pSFCChildWrite_EMX_SMFLDRN_CLOSED_TIME:      NOP 0;

      A "idbEMX4".f[#p.child.EMX_SMFLDRN].p.read.mc.modeAUTO;
      JCN _pSFCChildWrite_EMX_SMFLDRN_OPENED_TIME;
      L #p.write.EMX_SMFLDRN_OPENED_TIME;
      T "idbEMX4".f[#p.child.EMX_SMFLDRN].p.write.OPENED_TIME;
_pSFCChildWrite_EMX_SMFLDRN_OPENED_TIME:      NOP 0;

      A "idbEMX2".f[#p.child.EMX_TRANSFER1].p.read.mc.modeAUTO;
      JCN _pSFCChildWrite_EMX_TRANSFER1_FILL_FLZ;
      L #p.write.EMX_TRANSFER1_FILL_FLZ;
      T "idbEMX2".f[#p.child.EMX_TRANSFER1].p.write.FILL_FLZ;
_pSFCChildWrite_EMX_TRANSFER1_FILL_FLZ:      NOP 0;

      A "idbEMX2".f[#p.child.EMX_TRANSFER1].p.read.mc.modeAUTO;
      JCN _pSFCChildWrite_EMX_TRANSFER1_VESSEL_MX;
      L #p.write.EMX_TRANSFER1_VESSEL_MX;
      T "idbEMX2".f[#p.child.EMX_TRANSFER1].p.write.VESSEL_MX;
_pSFCChildWrite_EMX_TRANSFER1_VESSEL_MX:      NOP 0;

      A "idbEMX2".f[#p.child.EMX_TRANSFER2].p.read.mc.modeAUTO;
      JCN _pSFCChildWrite_EMX_TRANSFER2_FILL_FLZ;
      L #p.write.EMX_TRANSFER2_FILL_FLZ;
      T "idbEMX2".f[#p.child.EMX_TRANSFER2].p.write.FILL_FLZ;
_pSFCChildWrite_EMX_TRANSFER2_FILL_FLZ:      NOP 0;

      A "idbEMX2".f[#p.child.EMX_TRANSFER2].p.read.mc.modeAUTO;
      JCN _pSFCChildWrite_EMX_TRANSFER2_VESSEL_MX;
      L #p.write.EMX_TRANSFER2_VESSEL_MX;
      T "idbEMX2".f[#p.child.EMX_TRANSFER2].p.write.VESSEL_MX;
_pSFCChildWrite_EMX_TRANSFER2_VESSEL_MX:      NOP 0;

      A "idbEMA1".f[#p.child.EMA_VESSEL].p.read.mc.modeAUTO;
      JCN _pSFCChildWrite_EMA_VESSEL_RUNTIME_H;
      L #p.write.EMA_VESSEL_RUNTIME_H;
      T "idbEMA1".f[#p.child.EMA_VESSEL].p.write.RUNTIME_H;
_pSFCChildWrite_EMA_VESSEL_RUNTIME_H:      NOP 0;

      A "idbEMA1".f[#p.child.EMA_VESSEL].p.read.mc.modeAUTO;
      JCN _pSFCChildWrite_EMA_VESSEL_RUNTIME_M;
      L #p.write.EMA_VESSEL_RUNTIME_M;
      T "idbEMA1".f[#p.child.EMA_VESSEL].p.write.RUNTIME_M;
_pSFCChildWrite_EMA_VESSEL_RUNTIME_M:      NOP 0;

      A "idbEMA1".f[#p.child.EMA_VESSEL].p.read.mc.modeAUTO;
      JCN _pSFCChildWrite_EMA_VESSEL_RUNTIME_S;
      L #p.write.EMA_VESSEL_RUNTIME_S;
      T "idbEMA1".f[#p.child.EMA_VESSEL].p.write.RUNTIME_S;
_pSFCChildWrite_EMA_VESSEL_RUNTIME_S:      NOP 0;

      A "idbEMA1".f[#p.child.EMA_VESSEL].p.read.mc.modeAUTO;
      JCN _pSFCChildWrite_EMA_VESSEL_SETPOINT;
      L #p.write.EMA_VESSEL_SETPOINT;
      T "idbEMA1".f[#p.child.EMA_VESSEL].p.write.SETPOINT;
_pSFCChildWrite_EMA_VESSEL_SETPOINT:      NOP 0;

      A "idbEMC1".f[#p.child.EMC_GAS].p.read.mc.modeAUTO;
      JCN _pSFCChildWrite_EMC_GAS_MEDIUM_GAS;
      L #p.write.EMC_GAS_MEDIUM_GAS;
      T "idbEMC1".f[#p.child.EMC_GAS].p.write.MEDIUM_GAS;
_pSFCChildWrite_EMC_GAS_MEDIUM_GAS:      NOP 0;

      A "idbEMC1".f[#p.child.EMC_GAS].p.read.mc.modeAUTO;
      JCN _pSFCChildWrite_EMC_GAS_SETPOINT;
      L #p.write.EMC_GAS_SETPOINT;
      T "idbEMC1".f[#p.child.EMC_GAS].p.write.SETPOINT;
_pSFCChildWrite_EMC_GAS_SETPOINT:      NOP 0;

      A "idbEMC2".f[#p.child.EMC_WATER].p.read.mc.modeAUTO;
      JCN _pSFCChildWrite_EMC_WATER_MASS_CHARGE;
      L #p.write.EMC_WATER_MASS_CHARGE;
      T "idbEMC2".f[#p.child.EMC_WATER].p.write.MASS_CHARGE;
_pSFCChildWrite_EMC_WATER_MASS_CHARGE:      NOP 0;

      A "idbEMC2".f[#p.child.EMC_WATER].p.read.mc.modeAUTO;
      JCN _pSFCChildWrite_EMC_WATER_MEDIUM_LIQUID;
      L #p.write.EMC_WATER_MEDIUM_LIQUID;
      T "idbEMC2".f[#p.child.EMC_WATER].p.write.MEDIUM_LIQUID;
_pSFCChildWrite_EMC_WATER_MEDIUM_LIQUID:      NOP 0;

      A "idbEMC2".f[#p.child.EMC_WATER].p.read.mc.modeAUTO;
      JCN _pSFCChildWrite_EMC_WATER_RUNTIME;
      L #p.write.EMC_WATER_RUNTIME;
      T "idbEMC2".f[#p.child.EMC_WATER].p.write.RUNTIME;
_pSFCChildWrite_EMC_WATER_RUNTIME:      NOP 0;

      A "idbEMC2".f[#p.child.EMC_WATER].p.read.mc.modeAUTO;
      JCN _pSFCChildWrite_EMC_WATER_TIMEOUT;
      L #p.write.EMC_WATER_TIMEOUT;
      T "idbEMC2".f[#p.child.EMC_WATER].p.write.TIMEOUT;
_pSFCChildWrite_EMC_WATER_TIMEOUT:      NOP 0;

      A "idbEMM1".f[#p.child.EMM_VESSEL].p.read.mc.modeAUTO;
      JCN _pSFCChildWrite_EMM_VESSEL_SETTLING_TIME;
      L #p.write.EMM_VESSEL_SETTLING_TIME;
      T "idbEMM1".f[#p.child.EMM_VESSEL].p.write.SETTLING_TIME;
_pSFCChildWrite_EMM_VESSEL_SETTLING_TIME:      NOP 0;

      A "idbEMV2".f[#p.child.EMV_INLET].p.read.mc.modeAUTO;
      JCN _pSFCChildWrite_EMV_INLET_OPENED_TIME;
      L #p.write.EMV_INLET_OPENED_TIME;
      T "idbEMV2".f[#p.child.EMV_INLET].p.write.OPENED_TIME;
_pSFCChildWrite_EMV_INLET_OPENED_TIME:      NOP 0;

      A "idbEMT1".f[#p.child.EMT_HEX].p.read.mc.modeAUTO;
      JCN _pSFCChildWrite_EMT_HEX_SETPOINT;
      L #p.write.EMT_HEX_SETPOINT;
      T "idbEMT1".f[#p.child.EMT_HEX].p.write.SETPOINT;
_pSFCChildWrite_EMT_HEX_SETPOINT:      NOP 0;

      A "idbEMT1".f[#p.child.EMT_HEX].p.read.mc.modeAUTO;
      JCN _pSFCChildWrite_EMT_HEX_DRAIN_TIME;
      L #p.write.EMT_HEX_DRAIN_TIME;
      T "idbEMT1".f[#p.child.EMT_HEX].p.write.DRAIN_TIME;
_pSFCChildWrite_EMT_HEX_DRAIN_TIME:      NOP 0;


  //------------------------------------------------------------------------//
  // Write the boolean child parameters if no child mismatch:               //
  //------------------------------------------------------------------------//

_noCommandOnChildMismatch:      NOP 0;


